LIN {X 0,Y 105.507,Z 842.039,A -85,B 0,C 180,E1 -26362.344,E2 -26362.344} C_VEL
LIN {X 0,Y 105.583,Z 840.616,A -85,B 0,C 180,E1 -26366.845,E2 -26366.845} C_VEL
LIN {X 0,Y 105.811,Z 839.235,A -85,B 0,C 180,E1 -26370,E2 -26370} C_VEL
LIN {X 0,Y 105.61,Z 835.784,A -85,B 0,C 180,E1 -26375.729,E2 -26375.729} C_VEL
LIN {X 0,Y 106.123,Z 831.156,A -85,B 0,C 180,E1 -26381.459,E2 -26381.459} C_VEL
LIN {X 0,Y 107.753,Z 824.08,A -85,B 0,C 180,E1 -26388.047,E2 -26388.047} C_VEL
LIN {X 0,Y 110.175,Z 816.366,A -85,B 0,C 180,E1 -26393.495,E2 -26393.495} C_VEL
LIN {X 0,Y 112.77,Z 808.397,A -85,B 0,C 180,E1 -26397.866,E2 -26397.866} C_VEL
LIN {X 0,Y 116.022,Z 799.047,A -85,B 0,C 180,E1 -26401.859,E2 -26401.859} C_VEL
LIN {X 0,Y 119.623,Z 788.064,A -85,B 0,C 180,E1 -26405.461,E2 -26405.461} C_VEL
LIN {X 0,Y 123.122,Z 776.115,A -85,B 0,C 180,E1 -26408.371,E2 -26408.371} C_VEL
LIN {X 0,Y 124.907,Z 768.802,A -85,B 0,C 180,E1 -26409.785,E2 -26409.785} C_VEL
LIN {X 0,Y 125.577,Z 763.379,A -85,B 0,C 180,E1 -26410.817,E2 -26410.817} C_VEL
LIN {X 0,Y 124.86,Z 754.314,A -85,B 0,C 180,E1 -26412.635,E2 -26412.635} C_VEL
LIN {X 0,Y 123.8,Z 745.016,A -85,B 0,C 180,E1 -26414.201,E2 -26414.201} C_VEL
LIN {X 0,Y 123.899,Z 739.222,A -85,B 0,C 180,E1 -26414.796,E2 -26414.796} C_VEL
LIN {X 0,Y 126.912,Z 703.597,A -85,B 0,C 180,E1 -26416.978,E2 -26416.978} C_VEL
LIN {X 0,Y 126.157,Z 693.57,A -85,B 0,C 180,E1 -26418.047,E2 -26418.047} C_VEL
LIN {X 0,Y 121.74,Z 679.502,A -85,B 0,C 180,E1 -26420.71,E2 -26420.71} C_VEL
LIN {X 0,Y 116.424,Z 665.324,A -85,B 0,C 180,E1 -26423.976,E2 -26423.976} C_VEL
LIN {X 0,Y 112.883,Z 657.742,A -85,B 0,C 180,E1 -26426.201,E2 -26426.201} C_VEL
LIN {X 0,Y 107.627,Z 649.272,A -85,B 0,C 180,E1 -26429.595,E2 -26429.595} C_VEL
LIN {X 0,Y 105.851,Z 646.479,A -85,B 0,C 180,E1 -26430.815,E2 -26430.815} C_VEL
LIN {X 0,Y 103.858,Z 643.285,A -85,B 0,C 180,E1 -26432.273,E2 -26432.273} C_VEL
LIN {X 0,Y 101.38,Z 640.128,A -85,B 0,C 180,E1 -26434.117,E2 -26434.117} C_VEL
LIN {X 0,Y 100.745,Z 637.925,A -85,B 0,C 180,E1 -26434.819,E2 -26434.819} C_VEL
LIN {X 0,Y 100.81,Z 637.922,A -85,B 0,C 180,E1 -26439.598,E2 -26439.598} C_VEL
LIN {X 0,Y 101.186,Z 637.873,A -85,B 0,C 180,E1 -26447.971,E2 -26447.971} C_VEL
LIN {X 0,Y 101.263,Z 637.855,A -85,B 0,C 180,E1 -26452.019,E2 -26452.019} C_VEL
LIN {X 0,Y 101.846,Z 637.775,A -85,B 0,C 180,E1 -26459.998,E2 -26459.998} C_VEL
LIN {X 0,Y 101.264,Z 637.869,A -85,B 0,C 180,E1 -26467.977,E2 -26467.977} C_VEL
LIN {X 0,Y 101.122,Z 637.858,A -85,B 0,C 180,E1 -26473.349,E2 -26473.349} C_VEL
LIN {X 0,Y 100.813,Z 637.923,A -85,B 0,C 180,E1 -26480.398,E2 -26480.398} C_VEL
LIN {X 0,Y 100.771,Z 637.901,A -85,B 0,C 180,E1 -26484.957,E2 -26484.957} C_VEL
LIN {X 0,Y 100.702,Z 637.938,A -85,B 0,C 180,E1 -26493.127,E2 -26493.127} C_VEL
LIN {X 0,Y 100.697,Z 637.919,A -85,B 0,C 180,E1 -26499.852,E2 -26499.852} C_VEL
LIN {X 0,Y 100.727,Z 637.934,A -85,B 0,C 180,E1 -26505.756,E2 -26505.756} C_VEL
LIN {X 0,Y 100.667,Z 637.925,A -85,B 0,C 180,E1 -26511.074,E2 -26511.074} C_VEL
LIN {X 0,Y 100.696,Z 637.935,A -85,B 0,C 180,E1 -26516.877,E2 -26516.877} C_VEL
LIN {X 0,Y 100.783,Z 637.928,A -85,B 0,C 180,E1 -26525.267,E2 -26525.267} C_VEL
LIN {X 0,Y 100.886,Z 638.058,A -85,B 0,C 180,E1 -26531.284,E2 -26531.284} C_VEL
LIN {X 0,Y 101.875,Z 640.799,A -85,B 0,C 180,E1 -26532.253,E2 -26532.253} C_VEL
LIN {X 0,Y 104.241,Z 643.451,A -85,B 0,C 180,E1 -26533.956,E2 -26533.956} C_VEL
LIN {X 0,Y 106.42,Z 646.692,A -85,B 0,C 180,E1 -26535.509,E2 -26535.509} C_VEL
LIN {X 0,Y 109.893,Z 651.957,A -85,B 0,C 180,E1 -26537.795,E2 -26537.795} C_VEL
LIN {X 0,Y 117.451,Z 664.633,A -85,B 0,C 180,E1 -26542.344,E2 -26542.344} C_VEL
LIN {X 0,Y 125.255,Z 682.339,A -85,B 0,C 180,E1 -26546.683,E2 -26546.683} C_VEL
LIN {X 0,Y 127.714,Z 688.733,A -85,B 0,C 180,E1 -26547.991,E2 -26547.991} C_VEL
LIN {X 0,Y 123.869,Z 730.785,A -85,B 0,C 180,E1 -26550.508,E2 -26550.508} C_VEL
LIN {X 0,Y 121.841,Z 745.154,A -85,B 0,C 180,E1 -26552.014,E2 -26552.014} C_VEL
LIN {X 0,Y 119.489,Z 756.549,A -85,B 0,C 180,E1 -26553.713,E2 -26553.713} C_VEL
LIN {X 0,Y 116.492,Z 768.644,A -85,B 0,C 180,E1 -26556.212,E2 -26556.212} C_VEL
LIN {X 0,Y 112.705,Z 781.046,A -85,B 0,C 180,E1 -26559.623,E2 -26559.623} C_VEL
LIN {X 0,Y 109.184,Z 791.561,A -85,B 0,C 180,E1 -26563.524,E2 -26563.524} C_VEL
LIN {X 0,Y 105.565,Z 801.658,A -85,B 0,C 180,E1 -26568.435,E2 -26568.435} C_VEL
LIN {X 0,Y 102.872,Z 809.142,A -85,B 0,C 180,E1 -26573.144,E2 -26573.144} C_VEL
LIN {X 0,Y 100.663,Z 815.792,A -85,B 0,C 180,E1 -26578.431,E2 -26578.431} C_VEL
LIN {X 0,Y 98.92,Z 821.873,A -85,B 0,C 180,E1 -26584.636,E2 -26584.636} C_VEL
LIN {X 0,Y 97.816,Z 827.335,A -85,B 0,C 180,E1 -26592.091,E2 -26592.091} C_VEL
LIN {X 0,Y 98.036,Z 831.381,A -85,B 0,C 180,E1 -26599.823,E2 -26599.823} C_VEL
LIN {X 0,Y 99.854,Z 833.955,A -85,B 0,C 180,E1 -26607.626,E2 -26607.626} C_VEL
LIN {X 0,Y 102.246,Z 834.975,A -85,B 0,C 180,E1 -26613.323,E2 -26613.323} C_VEL
LIN {X 0,Y 107.098,Z 835.004,A -85,B 0,C 180,E1 -26620.848,E2 -26620.848} C_VEL
LIN {X 0,Y 111.102,Z 834.19,A -85,B 0,C 180,E1 -26625.345,E2 -26625.345} C_VEL
LIN {X 0,Y 115.718,Z 832.693,A -85,B 0,C 180,E1 -26629.504,E2 -26629.504} C_VEL
LIN {X 0,Y 123.721,Z 829.106,A -85,B 0,C 180,E1 -26635.114,E2 -26635.114} C_VEL
LIN {X 0,Y 131.219,Z 824.778,A -85,B 0,C 180,E1 -26639.243,E2 -26639.243} C_VEL
LIN {X 0,Y 139.405,Z 819.061,A -85,B 0,C 180,E1 -26642.891,E2 -26642.891} C_VEL
LIN {X 0,Y 146.38,Z 813.354,A -85,B 0,C 180,E1 -26645.512,E2 -26645.512} C_VEL
LIN {X 0,Y 153.61,Z 806.471,A -85,B 0,C 180,E1 -26647.89,E2 -26647.89} C_VEL
LIN {X 0,Y 161.109,Z 798.113,A -85,B 0,C 180,E1 -26650.05,E2 -26650.05} C_VEL
LIN {X 0,Y 167.935,Z 789.141,A -85,B 0,C 180,E1 -26651.742,E2 -26651.742} C_VEL
LIN {X 0,Y 174.832,Z 778.191,A -85,B 0,C 180,E1 -26653.355,E2 -26653.355} C_VEL
LIN {X 0,Y 180.883,Z 766.378,A -85,B 0,C 180,E1 -26654.649,E2 -26654.649} C_VEL
LIN {X 0,Y 185.753,Z 754.041,A -85,B 0,C 180,E1 -26655.675,E2 -26655.675} C_VEL
LIN {X 0,Y 189.546,Z 741.072,A -85,B 0,C 180,E1 -26656.406,E2 -26656.406} C_VEL
LIN {X 0,Y 191.061,Z 734.083,A -85,B 0,C 180,E1 -26656.709,E2 -26656.709} C_VEL
LIN {X 0,Y 190.49,Z 732.621,A -85,B 0,C 180,E1 -26659.394,E2 -26659.394} C_VEL
LIN {X 0,Y 190.206,Z 732.592,A -85,B 0,C 180,E1 -26662.525,E2 -26662.525} C_VEL
LIN {X 0,Y 190.233,Z 735.09,A -85,B 0,C 180,E1 -26665.607,E2 -26665.607} C_VEL
LIN {X 0,Y 190.431,Z 736.832,A -85,B 0,C 180,E1 -26667.146,E2 -26667.146} C_VEL
LIN {X 0,Y 190.517,Z 737.806,A -85,B 0,C 180,E1 -26667.826,E2 -26667.826} C_VEL
LIN {X 0,Y 187.086,Z 751.386,A -85,B 0,C 180,E1 -26668.382,E2 -26668.382} C_VEL
LIN {X 0,Y 182.826,Z 763.398,A -85,B 0,C 180,E1 -26669.013,E2 -26669.013} C_VEL
LIN {X 0,Y 177.372,Z 775.257,A -85,B 0,C 180,E1 -26669.919,E2 -26669.919} C_VEL
LIN {X 0,Y 170.424,Z 787.344,A -85,B 0,C 180,E1 -26671.166,E2 -26671.166} C_VEL
LIN {X 0,Y 162.951,Z 798.092,A -85,B 0,C 180,E1 -26672.754,E2 -26672.754} C_VEL
LIN {X 0,Y 154.273,Z 808.469,A -85,B 0,C 180,E1 -26674.917,E2 -26674.917} C_VEL
LIN {X 0,Y 147.223,Z 815.602,A -85,B 0,C 180,E1 -26676.91,E2 -26676.91} C_VEL
LIN {X 0,Y 137.903,Z 823.753,A -85,B 0,C 180,E1 -26680.144,E2 -26680.144} C_VEL
LIN {X 0,Y 130.48,Z 829.369,A -85,B 0,C 180,E1 -26683.354,E2 -26683.354} C_VEL
LIN {X 0,Y 123.528,Z 833.895,A -85,B 0,C 180,E1 -26686.944,E2 -26686.944} C_VEL
LIN {X 0,Y 115.371,Z 838.364,A -85,B 0,C 180,E1 -26692.472,E2 -26692.472} C_VEL
LIN {X 0,Y 108.476,Z 841.336,A -85,B 0,C 180,E1 -26698.782,E2 -26698.782} C_VEL
LIN {X 0,Y 103.18,Z 842.778,A -85,B 0,C 180,E1 -26705.878,E2 -26705.878} C_VEL
LIN {X 0,Y 99.85,Z 842.798,A -85,B 0,C 180,E1 -26713.648,E2 -26713.648} C_VEL
LIN {X 0,Y 98.483,Z 841.375,A -85,B 0,C 180,E1 -26721.795,E2 -26721.795} C_VEL
LIN {X 0,Y 98.543,Z 839.693,A -85,B 0,C 180,E1 -26726.862,E2 -26726.862} C_VEL
LIN {X 0,Y 98.752,Z 838.329,A -85,B 0,C 180,E1 -26730,E2 -26730} C_VEL
LIN {X 0,Y 98.559,Z 834.707,A -85,B 0,C 180,E1 -26736.14,E2 -26736.14} C_VEL
LIN {X 0,Y 99.163,Z 829.901,A -85,B 0,C 180,E1 -26742.276,E2 -26742.276} C_VEL
LIN {X 0,Y 100.66,Z 823.745,A -85,B 0,C 180,E1 -26748.311,E2 -26748.311} C_VEL
LIN {X 0,Y 103.166,Z 816.036,A -85,B 0,C 180,E1 -26754.125,E2 -26754.125} C_VEL
LIN {X 0,Y 106.558,Z 806.291,A -85,B 0,C 180,E1 -26759.646,E2 -26759.646} C_VEL
LIN {X 0,Y 110.231,Z 796.046,A -85,B 0,C 180,E1 -26764.017,E2 -26764.017} C_VEL
LIN {X 0,Y 113.917,Z 785.002,A -85,B 0,C 180,E1 -26767.533,E2 -26767.533} C_VEL
LIN {X 0,Y 117.16,Z 774.095,A -85,B 0,C 180,E1 -26770.153,E2 -26770.153} C_VEL
LIN {X 0,Y 120.102,Z 762.182,A -85,B 0,C 180,E1 -26772.294,E2 -26772.294} C_VEL
LIN {X 0,Y 122.613,Z 748.643,A -85,B 0,C 180,E1 -26773.989,E2 -26773.989} C_VEL
LIN {X 0,Y 123.899,Z 739.222,A -85,B 0,C 180,E1 -26774.796,E2 -26774.796} C_VEL
LIN {X 0,Y 123.887,Z 733.426,A -85,B 0,C 180,E1 -26775.338,E2 -26775.338} C_VEL
LIN {X 0,Y 120.636,Z 714.621,A -85,B 0,C 180,E1 -26777.918,E2 -26777.918} C_VEL
LIN {X 0,Y 120.649,Z 708.81,A -85,B 0,C 180,E1 -26778.427,E2 -26778.427} C_VEL
LIN {X 0,Y 120.935,Z 703.551,A -85,B 0,C 180,E1 -26778.807,E2 -26778.807} C_VEL
LIN {X 0,Y 120.332,Z 695.575,A -85,B 0,C 180,E1 -26779.728,E2 -26779.728} C_VEL
LIN {X 0,Y 116.176,Z 682.158,A -85,B 0,C 180,E1 -26782.432,E2 -26782.432} C_VEL
LIN {X 0,Y 110.783,Z 667.555,A -85,B 0,C 180,E1 -26786.084,E2 -26786.084} C_VEL
LIN {X 0,Y 108.118,Z 661.9,A -85,B 0,C 180,E1 -26787.932,E2 -26787.932} C_VEL
LIN {X 0,Y 101.977,Z 651.808,A -85,B 0,C 180,E1 -26792.275,E2 -26792.275} C_VEL
LIN {X 0,Y 99.367,Z 647.874,A -85,B 0,C 180,E1 -26794.342,E2 -26794.342} C_VEL
LIN {X 0,Y 97.298,Z 644.843,A -85,B 0,C 180,E1 -26796.087,E2 -26796.087} C_VEL
LIN {X 0,Y 96.693,Z 643.761,A -85,B 0,C 180,E1 -26796.649,E2 -26796.649} C_VEL
LIN {X 0,Y 94.607,Z 641.473,A -85,B 0,C 180,E1 -26798.48,E2 -26798.48} C_VEL
LIN {X 0,Y 93.783,Z 638.795,A -85,B 0,C 180,E1 -26799.719,E2 -26799.719} C_VEL
LIN {X 0,Y 94.09,Z 638.764,A -85,B 0,C 180,E1 -26807.049,E2 -26807.049} C_VEL
LIN {X 0,Y 94.196,Z 638.732,A -85,B 0,C 180,E1 -26811.416,E2 -26811.416} C_VEL
LIN {X 0,Y 94.776,Z 638.654,A -85,B 0,C 180,E1 -26819.998,E2 -26819.998} C_VEL
LIN {X 0,Y 94.197,Z 638.747,A -85,B 0,C 180,E1 -26828.579,E2 -26828.579} C_VEL
LIN {X 0,Y 94.039,Z 638.739,A -85,B 0,C 180,E1 -26833.706,E2 -26833.706} C_VEL
LIN {X 0,Y 93.69,Z 638.801,A -85,B 0,C 180,E1 -26842.026,E2 -26842.026} C_VEL
LIN {X 0,Y 93.618,Z 638.792,A -85,B 0,C 180,E1 -26846.768,E2 -26846.768} C_VEL
LIN {X 0,Y 93.609,Z 638.815,A -85,B 0,C 180,E1 -26854.326,E2 -26854.326} C_VEL
LIN {X 0,Y 93.628,Z 638.819,A -85,B 0,C 180,E1 -26862.495,E2 -26862.495} C_VEL
LIN {X 0,Y 93.598,Z 638.802,A -85,B 0,C 180,E1 -26868.662,E2 -26868.662} C_VEL
LIN {X 0,Y 93.599,Z 638.825,A -85,B 0,C 180,E1 -26875.681,E2 -26875.681} C_VEL
LIN {X 0,Y 93.665,Z 638.818,A -85,B 0,C 180,E1 -26884.205,E2 -26884.205} C_VEL
LIN {X 0,Y 93.719,Z 638.857,A -85,B 0,C 180,E1 -26886.466,E2 -26886.466} C_VEL
LIN {X 0,Y 94.603,Z 641.463,A -85,B 0,C 180,E1 -26887.526,E2 -26887.526} C_VEL
LIN {X 0,Y 96.702,Z 643.724,A -85,B 0,C 180,E1 -26889.328,E2 -26889.328} C_VEL
LIN {X 0,Y 97.427,Z 644.758,A -85,B 0,C 180,E1 -26889.954,E2 -26889.954} C_VEL
LIN {X 0,Y 99.513,Z 647.872,A -85,B 0,C 180,E1 -26891.727,E2 -26891.727} C_VEL
LIN {X 0,Y 100.58,Z 649.179,A -85,B 0,C 180,E1 -26892.558,E2 -26892.558} C_VEL
LIN {X 0,Y 105.142,Z 655.973,A -85,B 0,C 180,E1 -26895.939,E2 -26895.939} C_VEL
LIN {X 0,Y 112.658,Z 668.93,A -85,B 0,C 180,E1 -26900.848,E2 -26900.848} C_VEL
LIN {X 0,Y 119.963,Z 685.957,A -85,B 0,C 180,E1 -26905.255,E2 -26905.255} C_VEL
LIN {X 0,Y 121.748,Z 691.098,A -85,B 0,C 180,E1 -26906.309,E2 -26906.309} C_VEL
LIN {X 0,Y 117.785,Z 731.396,A -85,B 0,C 180,E1 -26908.785,E2 -26908.785} C_VEL
LIN {X 0,Y 115.797,Z 744.729,A -85,B 0,C 180,E1 -26910.217,E2 -26910.217} C_VEL
LIN {X 0,Y 113.226,Z 756.797,A -85,B 0,C 180,E1 -26912.065,E2 -26912.065} C_VEL
LIN {X 0,Y 110.198,Z 768.519,A -85,B 0,C 180,E1 -26914.572,E2 -26914.572} C_VEL
LIN {X 0,Y 106.425,Z 780.27,A -85,B 0,C 180,E1 -26917.897,E2 -26917.897} C_VEL
LIN {X 0,Y 102.829,Z 790.679,A -85,B 0,C 180,E1 -26921.832,E2 -26921.832} C_VEL
LIN {X 0,Y 98.939,Z 801.026,A -85,B 0,C 180,E1 -26927.038,E2 -26927.038} C_VEL
LIN {X 0,Y 95.746,Z 809.537,A -85,B 0,C 180,E1 -26932.666,E2 -26932.666} C_VEL
LIN {X 0,Y 93.15,Z 817.199,A -85,B 0,C 180,E1 -26939.367,E2 -26939.367} C_VEL
LIN {X 0,Y 91.604,Z 822.513,A -85,B 0,C 180,E1 -26945.364,E2 -26945.364} C_VEL
LIN {X 0,Y 90.762,Z 826.881,A -85,B 0,C 180,E1 -26951.639,E2 -26951.639} C_VEL
LIN {X 0,Y 90.777,Z 830.425,A -85,B 0,C 180,E1 -26958.313,E2 -26958.313} C_VEL
LIN {X 0,Y 92.378,Z 833.555,A -85,B 0,C 180,E1 -26966.809,E2 -26966.809} C_VEL
LIN {X 0,Y 95.035,Z 835.066,A -85,B 0,C 180,E1 -26973.662,E2 -26973.662} C_VEL
LIN {X 0,Y 98.125,Z 835.577,A -85,B 0,C 180,E1 -26979.018,E2 -26979.018} C_VEL
LIN {X 0,Y 102.213,Z 835.342,A -85,B 0,C 180,E1 -26984.28,E2 -26984.28} C_VEL
LIN {X 0,Y 107.28,Z 834.296,A -85,B 0,C 180,E1 -26989.306,E2 -26989.306} C_VEL
LIN {X 0,Y 113.091,Z 832.418,A -85,B 0,C 180,E1 -26993.874,E2 -26993.874} C_VEL
LIN {X 0,Y 119.551,Z 829.672,A -85,B 0,C 180,E1 -26997.925,E2 -26997.925} C_VEL
LIN {X 0,Y 128.331,Z 824.95,A -85,B 0,C 180,E1 -27002.331,E2 -27002.331} C_VEL
LIN {X 0,Y 137.033,Z 819.188,A -85,B 0,C 180,E1 -27005.889,E2 -27005.889} C_VEL
LIN {X 0,Y 145.96,Z 812.026,A -85,B 0,C 180,E1 -27008.888,E2 -27008.888} C_VEL
LIN {X 0,Y 155.535,Z 802.716,A -85,B 0,C 180,E1 -27011.619,E2 -27011.619} C_VEL
LIN {X 0,Y 162.888,Z 794.206,A -85,B 0,C 180,E1 -27013.39,E2 -27013.39} C_VEL
LIN {X 0,Y 170.093,Z 784.173,A -85,B 0,C 180,E1 -27014.968,E2 -27014.968} C_VEL
LIN {X 0,Y 176.246,Z 773.773,A -85,B 0,C 180,E1 -27016.21,E2 -27016.21} C_VEL
LIN {X 0,Y 181.857,Z 762.003,A -85,B 0,C 180,E1 -27017.284,E2 -27017.284} C_VEL
LIN {X 0,Y 186.117,Z 750.546,A -85,B 0,C 180,E1 -27018.084,E2 -27018.084} C_VEL
LIN {X 0,Y 189.08,Z 739.923,A -85,B 0,C 180,E1 -27018.664,E2 -27018.664} C_VEL
LIN {X 0,Y 188.982,Z 739.555,A -85,B 0,C 180,E1 -27019.555,E2 -27019.555} C_VEL
LIN {X 0,Y 188.748,Z 739.568,A -85,B 0,C 180,E1 -27022.51,E2 -27022.51} C_VEL
LIN {X 0,Y 188.622,Z 742.467,A -85,B 0,C 180,E1 -27025.859,E2 -27025.859} C_VEL
LIN {X 0,Y 184.48,Z 756.22,A -85,B 0,C 180,E1 -27026.42,E2 -27026.42} C_VEL
LIN {X 0,Y 179.622,Z 768.209,A -85,B 0,C 180,E1 -27027.113,E2 -27027.113} C_VEL
LIN {X 0,Y 173.247,Z 780.405,A -85,B 0,C 180,E1 -27028.079,E2 -27028.079} C_VEL
LIN {X 0,Y 166.211,Z 791.358,A -85,B 0,C 180,E1 -27029.299,E2 -27029.299} C_VEL
LIN {X 0,Y 159.316,Z 800.338,A -85,B 0,C 180,E1 -27030.662,E2 -27030.662} C_VEL
LIN {X 0,Y 150.398,Z 810.137,A -85,B 0,C 180,E1 -27032.743,E2 -27032.743} C_VEL
LIN {X 0,Y 141.745,Z 818.173,A -85,B 0,C 180,E1 -27035.107,E2 -27035.107} C_VEL
LIN {X 0,Y 133.482,Z 824.729,A -85,B 0,C 180,E1 -27037.838,E2 -27037.838} C_VEL
LIN {X 0,Y 125.751,Z 830.037,A -85,B 0,C 180,E1 -27041.021,E2 -27041.021} C_VEL
LIN {X 0,Y 118.45,Z 834.317,A -85,B 0,C 180,E1 -27044.604,E2 -27044.604} C_VEL
LIN {X 0,Y 109.815,Z 838.571,A -85,B 0,C 180,E1 -27050.21,E2 -27050.21} C_VEL
LIN {X 0,Y 102.46,Z 841.237,A -85,B 0,C 180,E1 -27056.72,E2 -27056.72} C_VEL
LIN {X 0,Y 96.739,Z 842.474,A -85,B 0,C 180,E1 -27064.159,E2 -27064.159} C_VEL
LIN {X 0,Y 93.023,Z 842.298,A -85,B 0,C 180,E1 -27072.41,E2 -27072.41} C_VEL
LIN {X 0,Y 91.467,Z 840.637,A -85,B 0,C 180,E1 -27081.16,E2 -27081.16} C_VEL
LIN {X 0,Y 91.509,Z 838.797,A -85,B 0,C 180,E1 -27086.809,E2 -27086.809} C_VEL
LIN {X 0,Y 91.695,Z 837.408,A -85,B 0,C 180,E1 -27090,E2 -27090} C_VEL
LIN {X 0,Y 91.519,Z 833.589,A -85,B 0,C 180,E1 -27096.614,E2 -27096.614} C_VEL
LIN {X 0,Y 92.239,Z 828.574,A -85,B 0,C 180,E1 -27103.213,E2 -27103.213} C_VEL
LIN {X 0,Y 93.948,Z 822.181,A -85,B 0,C 180,E1 -27109.671,E2 -27109.671} C_VEL
LIN {X 0,Y 96.695,Z 814.135,A -85,B 0,C 180,E1 -27115.854,E2 -27115.854} C_VEL
LIN {X 0,Y 99.745,Z 805.915,A -85,B 0,C 180,E1 -27120.719,E2 -27120.719} C_VEL
LIN {X 0,Y 103.507,Z 795.936,A -85,B 0,C 180,E1 -27125.242,E2 -27125.242} C_VEL
LIN {X 0,Y 107.442,Z 784.692,A -85,B 0,C 180,E1 -27129.019,E2 -27129.019} C_VEL
LIN {X 0,Y 110.827,Z 773.799,A -85,B 0,C 180,E1 -27131.746,E2 -27131.746} C_VEL
LIN {X 0,Y 114.175,Z 760.719,A -85,B 0,C 180,E1 -27134.133,E2 -27134.133} C_VEL
LIN {X 0,Y 116.664,Z 747.345,A -85,B 0,C 180,E1 -27135.826,E2 -27135.826} C_VEL
LIN {X 0,Y 118.395,Z 733.513,A -85,B 0,C 180,E1 -27136.919,E2 -27136.919} C_VEL
LIN {X 0,Y 120.649,Z 708.81,A -85,B 0,C 180,E1 -27138.427,E2 -27138.427} C_VEL
LIN {X 0,Y 120.572,Z 705.009,A -85,B 0,C 180,E1 -27138.795,E2 -27138.795} C_VEL
LIN {X 0,Y 119.745,Z 701.405,A -85,B 0,C 180,E1 -27139.393,E2 -27139.393} C_VEL
LIN {X 0,Y 118.4,Z 698.014,A -85,B 0,C 180,E1 -27140.164,E2 -27140.164} C_VEL
LIN {X 0,Y 110.38,Z 683.673,A -85,B 0,C 180,E1 -27144.553,E2 -27144.553} C_VEL
LIN {X 0,Y 109.72,Z 681.909,A -85,B 0,C 180,E1 -27145.018,E2 -27145.018} C_VEL
LIN {X 0,Y 104.964,Z 669.063,A -85,B 0,C 180,E1 -27148.633,E2 -27148.633} C_VEL
LIN {X 0,Y 99.77,Z 659.846,A -85,B 0,C 180,E1 -27152.528,E2 -27152.528} C_VEL
LIN {X 0,Y 95.437,Z 652.984,A -85,B 0,C 180,E1 -27156.218,E2 -27156.218} C_VEL
LIN {X 0,Y 92.964,Z 649.251,A -85,B 0,C 180,E1 -27158.517,E2 -27158.517} C_VEL
LIN {X 0,Y 90.71,Z 646.109,A -85,B 0,C 180,E1 -27160.773,E2 -27160.773} C_VEL
LIN {X 0,Y 90.069,Z 644.86,A -85,B 0,C 180,E1 -27161.516,E2 -27161.516} C_VEL
LIN {X 0,Y 87.854,Z 642.603,A -85,B 0,C 180,E1 -27163.905,E2 -27163.905} C_VEL
LIN {X 0,Y 86.916,Z 639.892,A -85,B 0,C 180,E1 -27165.312,E2 -27165.312} C_VEL
LIN {X 0,Y 86.969,Z 639.655,A -85,B 0,C 180,E1 -27165.968,E2 -27165.968} C_VEL
LIN {X 0,Y 87.105,Z 639.614,A -85,B 0,C 180,E1 -27170.711,E2 -27170.711} C_VEL
LIN {X 0,Y 87.706,Z 639.534,A -85,B 0,C 180,E1 -27179.998,E2 -27179.998} C_VEL
LIN {X 0,Y 87.105,Z 639.625,A -85,B 0,C 180,E1 -27189.284,E2 -27189.284} C_VEL
LIN {X 0,Y 86.948,Z 639.623,A -85,B 0,C 180,E1 -27194.085,E2 -27194.085} C_VEL
LIN {X 0,Y 86.659,Z 639.687,A -85,B 0,C 180,E1 -27198.927,E2 -27198.927} C_VEL
LIN {X 0,Y 86.581,Z 639.668,A -85,B 0,C 180,E1 -27206.763,E2 -27206.763} C_VEL
LIN {X 0,Y 86.534,Z 639.683,A -85,B 0,C 180,E1 -27215.693,E2 -27215.693} C_VEL
LIN {X 0,Y 86.553,Z 639.702,A -85,B 0,C 180,E1 -27223.049,E2 -27223.049} C_VEL
LIN {X 0,Y 86.505,Z 639.683,A -85,B 0,C 180,E1 -27229.463,E2 -27229.463} C_VEL
LIN {X 0,Y 86.545,Z 639.705,A -85,B 0,C 180,E1 -27235.359,E2 -27235.359} C_VEL
LIN {X 0,Y 86.494,Z 639.814,A -85,B 0,C 180,E1 -27240.238,E2 -27240.238} C_VEL
LIN {X 0,Y 87.41,Z 642.419,A -85,B 0,C 180,E1 -27241.619,E2 -27241.619} C_VEL
LIN {X 0,Y 89.42,Z 644.526,A -85,B 0,C 180,E1 -27243.853,E2 -27243.853} C_VEL
LIN {X 0,Y 90.277,Z 645.19,A -85,B 0,C 180,E1 -27244.708,E2 -27244.708} C_VEL
LIN {X 0,Y 92.207,Z 648.436,A -85,B 0,C 180,E1 -27246.795,E2 -27246.795} C_VEL
LIN {X 0,Y 93.86,Z 650.398,A -85,B 0,C 180,E1 -27248.323,E2 -27248.323} C_VEL
LIN {X 0,Y 97.533,Z 655.716,A -85,B 0,C 180,E1 -27251.529,E2 -27251.529} C_VEL
LIN {X 0,Y 100.981,Z 660.89,A -85,B 0,C 180,E1 -27254.292,E2 -27254.292} C_VEL
LIN {X 0,Y 107.991,Z 673.429,A -85,B 0,C 180,E1 -27259.274,E2 -27259.274} C_VEL
LIN {X 0,Y 114.654,Z 689.462,A -85,B 0,C 180,E1 -27263.703,E2 -27263.703} C_VEL
LIN {X 0,Y 115.771,Z 692.545,A -85,B 0,C 180,E1 -27264.411,E2 -27264.411} C_VEL
LIN {X 0,Y 111.744,Z 732.209,A -85,B 0,C 180,E1 -27266.958,E2 -27266.958} C_VEL
LIN {X 0,Y 109.669,Z 745.169,A -85,B 0,C 180,E1 -27268.393,E2 -27268.393} C_VEL
LIN {X 0,Y 106.957,Z 757.273,A -85,B 0,C 180,E1 -27270.312,E2 -27270.312} C_VEL
LIN {X 0,Y 103.775,Z 768.917,A -85,B 0,C 180,E1 -27272.901,E2 -27272.901} C_VEL
LIN {X 0,Y 99.81,Z 780.816,A -85,B 0,C 180,E1 -27276.439,E2 -27276.439} C_VEL
LIN {X 0,Y 96.046,Z 791.091,A -85,B 0,C 180,E1 -27280.54,E2 -27280.54} C_VEL
LIN {X 0,Y 91.938,Z 801.492,A -85,B 0,C 180,E1 -27286.114,E2 -27286.114} C_VEL
LIN {X 0,Y 88.48,Z 810.434,A -85,B 0,C 180,E1 -27292.524,E2 -27292.524} C_VEL
LIN {X 0,Y 85.946,Z 817.595,A -85,B 0,C 180,E1 -27299.381,E2 -27299.381} C_VEL
LIN {X 0,Y 84.406,Z 822.712,A -85,B 0,C 180,E1 -27305.65,E2 -27305.65} C_VEL
LIN {X 0,Y 83.639,Z 826.97,A -85,B 0,C 180,E1 -27312.238,E2 -27312.238} C_VEL
LIN {X 0,Y 84.082,Z 831.492,A -85,B 0,C 180,E1 -27321.755,E2 -27321.755} C_VEL
LIN {X 0,Y 86.492,Z 834.395,A -85,B 0,C 180,E1 -27330.824,E2 -27330.824} C_VEL
LIN {X 0,Y 90.405,Z 835.764,A -85,B 0,C 180,E1 -27338.883,E2 -27338.883} C_VEL
LIN {X 0,Y 94.704,Z 835.958,A -85,B 0,C 180,E1 -27344.733,E2 -27344.733} C_VEL
LIN {X 0,Y 102.172,Z 834.842,A -85,B 0,C 180,E1 -27352.095,E2 -27352.095} C_VEL
LIN {X 0,Y 107.791,Z 833.297,A -85,B 0,C 180,E1 -27356.264,E2 -27356.264} C_VEL
LIN {X 0,Y 116.995,Z 829.686,A -85,B 0,C 180,E1 -27361.611,E2 -27361.611} C_VEL
LIN {X 0,Y 127.227,Z 824.381,A -85,B 0,C 180,E1 -27366.126,E2 -27366.126} C_VEL
LIN {X 0,Y 135.199,Z 819.222,A -85,B 0,C 180,E1 -27369.016,E2 -27369.016} C_VEL
LIN {X 0,Y 145.246,Z 811.395,A -85,B 0,C 180,E1 -27372.031,E2 -27372.031} C_VEL
LIN {X 0,Y 154.179,Z 802.972,A -85,B 0,C 180,E1 -27374.29,E2 -27374.29} C_VEL
LIN {X 0,Y 161.612,Z 794.605,A -85,B 0,C 180,E1 -27375.894,E2 -27375.894} C_VEL
LIN {X 0,Y 169.444,Z 783.961,A -85,B 0,C 180,E1 -27377.457,E2 -27377.457} C_VEL
LIN {X 0,Y 176.022,Z 773.076,A -85,B 0,C 180,E1 -27378.629,E2 -27378.629} C_VEL
LIN {X 0,Y 181.681,Z 761.35,A -85,B 0,C 180,E1 -27379.615,E2 -27379.615} C_VEL
LIN {X 0,Y 185.783,Z 750.33,A -85,B 0,C 180,E1 -27380.313,E2 -27380.313} C_VEL
LIN {X 0,Y 187.019,Z 746.321,A -85,B 0,C 180,E1 -27380.577,E2 -27380.577} C_VEL
LIN {X 0,Y 186.93,Z 746.359,A -85,B 0,C 180,E1 -27382.085,E2 -27382.085} C_VEL
LIN {X 0,Y 186.816,Z 746.986,A -85,B 0,C 180,E1 -27382.965,E2 -27382.965} C_VEL
LIN {X 0,Y 186.596,Z 748.107,A -85,B 0,C 180,E1 -27383.898,E2 -27383.898} C_VEL
LIN {X 0,Y 182.032,Z 760.983,A -85,B 0,C 180,E1 -27384.44,E2 -27384.44} C_VEL
LIN {X 0,Y 176.601,Z 772.704,A -85,B 0,C 180,E1 -27385.132,E2 -27385.132} C_VEL
LIN {X 0,Y 169.301,Z 785.058,A -85,B 0,C 180,E1 -27386.146,E2 -27386.146} C_VEL
LIN {X 0,Y 162.156,Z 795.047,A -85,B 0,C 180,E1 -27387.319,E2 -27387.319} C_VEL
LIN {X 0,Y 154.375,Z 804.217,A -85,B 0,C 180,E1 -27388.796,E2 -27388.796} C_VEL
LIN {X 0,Y 145.24,Z 813.218,A -85,B 0,C 180,E1 -27390.809,E2 -27390.809} C_VEL
LIN {X 0,Y 136.407,Z 820.55,A -85,B 0,C 180,E1 -27393.153,E2 -27393.153} C_VEL
LIN {X 0,Y 126.552,Z 827.482,A -85,B 0,C 180,E1 -27396.368,E2 -27396.368} C_VEL
LIN {X 0,Y 118.606,Z 832.183,A -85,B 0,C 180,E1 -27399.619,E2 -27399.619} C_VEL
LIN {X 0,Y 111.188,Z 835.883,A -85,B 0,C 180,E1 -27403.375,E2 -27403.375} C_VEL
LIN {X 0,Y 104.245,Z 838.768,A -85,B 0,C 180,E1 -27407.871,E2 -27407.871} C_VEL
LIN {X 0,Y 96.595,Z 841.138,A -85,B 0,C 180,E1 -27414.406,E2 -27414.406} C_VEL
LIN {X 0,Y 90.4,Z 842.159,A -85,B 0,C 180,E1 -27422.196,E2 -27422.196} C_VEL
LIN {X 0,Y 86.256,Z 841.716,A -85,B 0,C 180,E1 -27430.979,E2 -27430.979} C_VEL
LIN {X 0,Y 84.477,Z 839.863,A -85,B 0,C 180,E1 -27440.422,E2 -27440.422} C_VEL
LIN {X 0,Y 84.476,Z 837.799,A -85,B 0,C 180,E1 -27446.742,E2 -27446.742} C_VEL
LIN {X 0,Y 84.64,Z 836.432,A -85,B 0,C 180,E1 -27450,E2 -27450} C_VEL
LIN {X 0,Y 84.509,Z 832.427,A -85,B 0,C 180,E1 -27457.166,E2 -27457.166} C_VEL
LIN {X 0,Y 85.594,Z 826.158,A -85,B 0,C 180,E1 -27465.477,E2 -27465.477} C_VEL
LIN {X 0,Y 87.746,Z 819.266,A -85,B 0,C 180,E1 -27472.361,E2 -27472.361} C_VEL
LIN {X 0,Y 90.337,Z 812.178,A -85,B 0,C 180,E1 -27477.825,E2 -27477.825} C_VEL
LIN {X 0,Y 93.725,Z 803.621,A -85,B 0,C 180,E1 -27482.931,E2 -27482.931} C_VEL
LIN {X 0,Y 97.808,Z 793.107,A -85,B 0,C 180,E1 -27487.637,E2 -27487.637} C_VEL
LIN {X 0,Y 101.53,Z 782.738,A -85,B 0,C 180,E1 -27491.116,E2 -27491.116} C_VEL
LIN {X 0,Y 105.136,Z 771.513,A -85,B 0,C 180,E1 -27493.909,E2 -27493.909} C_VEL
LIN {X 0,Y 108.357,Z 758.907,A -85,B 0,C 180,E1 -27496.182,E2 -27496.182} C_VEL
LIN {X 0,Y 110.833,Z 745.918,A -85,B 0,C 180,E1 -27497.825,E2 -27497.825} C_VEL
LIN {X 0,Y 112.49,Z 732.469,A -85,B 0,C 180,E1 -27498.891,E2 -27498.891} C_VEL
LIN {X 0,Y 115.06,Z 704.596,A -85,B 0,C 180,E1 -27500.679,E2 -27500.679} C_VEL
LIN {X 0,Y 114.624,Z 697.867,A -85,B 0,C 180,E1 -27501.483,E2 -27501.483} C_VEL
LIN {X 0,Y 110.368,Z 683.84,A -85,B 0,C 180,E1 -27504.54,E2 -27504.54} C_VEL
LIN {X 0,Y 109.72,Z 681.909,A -85,B 0,C 180,E1 -27505.018,E2 -27505.018} C_VEL
LIN {X 0,Y 107.504,Z 677.233,A -85,B 0,C 180,E1 -27506.514,E2 -27506.514} C_VEL
LIN {X 0,Y 104.576,Z 673.318,A -85,B 0,C 180,E1 -27508.345,E2 -27508.345} C_VEL
LIN {X 0,Y 94.062,Z 661.932,A -85,B 0,C 180,E1 -27515.877,E2 -27515.877} C_VEL
LIN {X 0,Y 89.49,Z 654.791,A -85,B 0,C 180,E1 -27520.351,E2 -27520.351} C_VEL
LIN {X 0,Y 87.111,Z 651.088,A -85,B 0,C 180,E1 -27523.068,E2 -27523.068} C_VEL
LIN {X 0,Y 84.527,Z 647.786,A -85,B 0,C 180,E1 -27526.25,E2 -27526.25} C_VEL
LIN {X 0,Y 83.55,Z 645.868,A -85,B 0,C 180,E1 -27527.674,E2 -27527.674} C_VEL
LIN {X 0,Y 81.381,Z 643.831,A -85,B 0,C 180,E1 -27530.679,E2 -27530.679} C_VEL
LIN {X 0,Y 80.239,Z 641.5,A -85,B 0,C 180,E1 -27532.764,E2 -27532.764} C_VEL
LIN {X 0,Y 80.055,Z 640.503,A -85,B 0,C 180,E1 -27533.381,E2 -27533.381} C_VEL
LIN {X 0,Y 80.637,Z 640.414,A -85,B 0,C 180,E1 -27539.997,E2 -27539.997} C_VEL
LIN {X 0,Y 79.99,Z 640.501,A -85,B 0,C 180,E1 -27550.118,E2 -27550.118} C_VEL
LIN {X 0,Y 79.763,Z 640.522,A -85,B 0,C 180,E1 -27555.325,E2 -27555.325} C_VEL
LIN {X 0,Y 79.519,Z 640.573,A -85,B 0,C 180,E1 -27560.7,E2 -27560.7} C_VEL
LIN {X 0,Y 79.48,Z 640.557,A -85,B 0,C 180,E1 -27567.843,E2 -27567.843} C_VEL
LIN {X 0,Y 79.444,Z 640.558,A -85,B 0,C 180,E1 -27577.235,E2 -27577.235} C_VEL
LIN {X 0,Y 79.463,Z 640.585,A -85,B 0,C 180,E1 -27585.032,E2 -27585.032} C_VEL
LIN {X 0,Y 79.42,Z 640.719,A -85,B 0,C 180,E1 -27591.813,E2 -27591.813} C_VEL
LIN {X 0,Y 80.226,Z 643.043,A -85,B 0,C 180,E1 -27593.577,E2 -27593.577} C_VEL
LIN {X 0,Y 82.617,Z 645.624,A -85,B 0,C 180,E1 -27597.23,E2 -27597.23} C_VEL
LIN {X 0,Y 83.471,Z 646.222,A -85,B 0,C 180,E1 -27598.33,E2 -27598.33} C_VEL
LIN {X 0,Y 85.083,Z 649.145,A -85,B 0,C 180,E1 -27600.604,E2 -27600.604} C_VEL
LIN {X 0,Y 87.31,Z 651.486,A -85,B 0,C 180,E1 -27603.166,E2 -27603.166} C_VEL
LIN {X 0,Y 89.77,Z 655.097,A -85,B 0,C 180,E1 -27605.927,E2 -27605.927} C_VEL
LIN {X 0,Y 95.39,Z 663.348,A -85,B 0,C 180,E1 -27611.215,E2 -27611.215} C_VEL
LIN {X 0,Y 102.913,Z 676.765,A -85,B 0,C 180,E1 -27617.255,E2 -27617.255} C_VEL
LIN {X 0,Y 109.463,Z 692.987,A -85,B 0,C 180,E1 -27622.014,E2 -27622.014} C_VEL
LIN {X 0,Y 109.867,Z 694.16,A -85,B 0,C 180,E1 -27622.304,E2 -27622.304} C_VEL
LIN {X 0,Y 105.834,Z 732.868,A -85,B 0,C 180,E1 -27624.905,E2 -27624.905} C_VEL
LIN {X 0,Y 103.663,Z 745.613,A -85,B 0,C 180,E1 -27626.356,E2 -27626.356} C_VEL
LIN {X 0,Y 100.62,Z 758.485,A -85,B 0,C 180,E1 -27628.499,E2 -27628.499} C_VEL
LIN {X 0,Y 96.777,Z 771.356,A -85,B 0,C 180,E1 -27631.565,E2 -27631.565} C_VEL
LIN {X 0,Y 92.821,Z 782.533,A -85,B 0,C 180,E1 -27635.217,E2 -27635.217} C_VEL
LIN {X 0,Y 88.794,Z 792.677,A -85,B 0,C 180,E1 -27639.683,E2 -27639.683} C_VEL
LIN {X 0,Y 84.58,Z 802.806,A -85,B 0,C 180,E1 -27645.667,E2 -27645.667} C_VEL
LIN {X 0,Y 81.563,Z 810.236,A -85,B 0,C 180,E1 -27651.481,E2 -27651.481} C_VEL
LIN {X 0,Y 78.978,Z 817.221,A -85,B 0,C 180,E1 -27658.553,E2 -27658.553} C_VEL
LIN {X 0,Y 77.02,Z 823.72,A -85,B 0,C 180,E1 -27667.31,E2 -27667.31} C_VEL
LIN {X 0,Y 76.458,Z 827.978,A -85,B 0,C 180,E1 -27674.817,E2 -27674.817} C_VEL
LIN {X 0,Y 77.467,Z 832.162,A -85,B 0,C 180,E1 -27684.734,E2 -27684.734} C_VEL
LIN {X 0,Y 80.441,Z 834.861,A -85,B 0,C 180,E1 -27694.1,E2 -27694.1} C_VEL
LIN {X 0,Y 83.677,Z 835.938,A -85,B 0,C 180,E1 -27700.372,E2 -27700.372} C_VEL
LIN {X 0,Y 87.888,Z 836.361,A -85,B 0,C 180,E1 -27706.122,E2 -27706.122} C_VEL
LIN {X 0,Y 92.738,Z 836.122,A -85,B 0,C 180,E1 -27711.285,E2 -27711.285} C_VEL
LIN {X 0,Y 98.615,Z 835.129,A -85,B 0,C 180,E1 -27716.124,E2 -27716.124} C_VEL
LIN {X 0,Y 108.22,Z 832.398,A -85,B 0,C 180,E1 -27722.141,E2 -27722.141} C_VEL
LIN {X 0,Y 118.261,Z 828.206,A -85,B 0,C 180,E1 -27726.828,E2 -27726.828} C_VEL
LIN {X 0,Y 128.714,Z 822.59,A -85,B 0,C 180,E1 -27730.64,E2 -27730.64} C_VEL
LIN {X 0,Y 137.119,Z 817.009,A -85,B 0,C 180,E1 -27733.141,E2 -27733.141} C_VEL
LIN {X 0,Y 145.761,Z 810.165,A -85,B 0,C 180,E1 -27735.358,E2 -27735.358} C_VEL
LIN {X 0,Y 154.568,Z 801.843,A -85,B 0,C 180,E1 -27737.289,E2 -27737.289} C_VEL
LIN {X 0,Y 163.469,Z 791.686,A -85,B 0,C 180,E1 -27738.947,E2 -27738.947} C_VEL
LIN {X 0,Y 170.607,Z 781.773,A -85,B 0,C 180,E1 -27740.172,E2 -27740.172} C_VEL
LIN {X 0,Y 176.972,Z 770.886,A -85,B 0,C 180,E1 -27741.192,E2 -27741.192} C_VEL
LIN {X 0,Y 181.833,Z 760.595,A -85,B 0,C 180,E1 -27741.937,E2 -27741.937} C_VEL
LIN {X 0,Y 182.095,Z 759.994,A -85,B 0,C 180,E1 -27742.141,E2 -27742.141} C_VEL
LIN {X 0,Y 176.767,Z 771.468,A -85,B 0,C 180,E1 -27742.733,E2 -27742.733} C_VEL
LIN {X 0,Y 169.657,Z 783.547,A -85,B 0,C 180,E1 -27743.581,E2 -27743.581} C_VEL
LIN {X 0,Y 162.326,Z 793.69,A -85,B 0,C 180,E1 -27744.607,E2 -27744.607} C_VEL
LIN {X 0,Y 154.312,Z 802.96,A -85,B 0,C 180,E1 -27745.911,E2 -27745.911} C_VEL
LIN {X 0,Y 144.886,Z 812.122,A -85,B 0,C 180,E1 -27747.72,E2 -27747.72} C_VEL
LIN {X 0,Y 135.69,Z 819.594,A -85,B 0,C 180,E1 -27749.826,E2 -27749.826} C_VEL
LIN {X 0,Y 125.354,Z 826.594,A -85,B 0,C 180,E1 -27752.759,E2 -27752.759} C_VEL
LIN {X 0,Y 116.977,Z 831.35,A -85,B 0,C 180,E1 -27755.8,E2 -27755.8} C_VEL
LIN {X 0,Y 108.971,Z 835.161,A -85,B 0,C 180,E1 -27759.294,E2 -27759.294} C_VEL
LIN {X 0,Y 99.311,Z 838.823,A -85,B 0,C 180,E1 -27764.955,E2 -27764.955} C_VEL
LIN {X 0,Y 90.91,Z 841.013,A -85,B 0,C 180,E1 -27771.798,E2 -27771.798} C_VEL
LIN {X 0,Y 84.183,Z 841.759,A -85,B 0,C 180,E1 -27779.941,E2 -27779.941} C_VEL
LIN {X 0,Y 79.554,Z 841.121,A -85,B 0,C 180,E1 -27789.307,E2 -27789.307} C_VEL
LIN {X 0,Y 77.512,Z 839.063,A -85,B 0,C 180,E1 -27799.552,E2 -27799.552} C_VEL
LIN {X 0,Y 77.448,Z 836.774,A -85,B 0,C 180,E1 -27806.602,E2 -27806.602} C_VEL
LIN {X 0,Y 77.597,Z 835.362,A -85,B 0,C 180,E1 -27810,E2 -27810} C_VEL
LIN {X 0,Y 77.517,Z 831.154,A -85,B 0,C 180,E1 -27817.816,E2 -27817.816} C_VEL
LIN {X 0,Y 78.514,Z 825.689,A -85,B 0,C 180,E1 -27825.577,E2 -27825.577} C_VEL
LIN {X 0,Y 80.74,Z 818.802,A -85,B 0,C 180,E1 -27833.06,E2 -27833.06} C_VEL
LIN {X 0,Y 83.468,Z 811.718,A -85,B 0,C 180,E1 -27838.956,E2 -27838.956} C_VEL
LIN {X 0,Y 87.051,Z 803.136,A -85,B 0,C 180,E1 -27844.411,E2 -27844.411} C_VEL
LIN {X 0,Y 91.033,Z 793.39,A -85,B 0,C 180,E1 -27849.064,E2 -27849.064} C_VEL
LIN {X 0,Y 95.267,Z 782.191,A -85,B 0,C 180,E1 -27853.029,E2 -27853.029} C_VEL
LIN {X 0,Y 99.047,Z 770.898,A -85,B 0,C 180,E1 -27855.924,E2 -27855.924} C_VEL
LIN {X 0,Y 102.403,Z 758.202,A -85,B 0,C 180,E1 -27858.274,E2 -27858.274} C_VEL
LIN {X 0,Y 105,Z 745.081,A -85,B 0,C 180,E1 -27859.954,E2 -27859.954} C_VEL
LIN {X 0,Y 106.91,Z 729.875,A -85,B 0,C 180,E1 -27861.129,E2 -27861.129} C_VEL
LIN {X 0,Y 109.277,Z 705.445,A -85,B 0,C 180,E1 -27862.739,E2 -27862.739} C_VEL
LIN {X 0,Y 108.9,Z 699.726,A -85,B 0,C 180,E1 -27863.488,E2 -27863.488} C_VEL
LIN {X 0,Y 104.993,Z 686.378,A -85,B 0,C 180,E1 -27866.658,E2 -27866.658} C_VEL
LIN {X 0,Y 100.292,Z 673.232,A -85,B 0,C 180,E1 -27870.532,E2 -27870.532} C_VEL
LIN {X 0,Y 95.738,Z 664.824,A -85,B 0,C 180,E1 -27874.348,E2 -27874.348} C_VEL
LIN {X 0,Y 94.062,Z 661.932,A -85,B 0,C 180,E1 -27875.877,E2 -27875.877} C_VEL
LIN {X 0,Y 92.07,Z 659.911,A -85,B 0,C 180,E1 -27877.561,E2 -27877.561} C_VEL
LIN {X 0,Y 88.27,Z 658.103,A -85,B 0,C 180,E1 -27880.836,E2 -27880.836} C_VEL
LIN {X 0,Y 83.89,Z 656.302,A -85,B 0,C 180,E1 -27885.256,E2 -27885.256} C_VEL
LIN {X 0,Y 82.646,Z 655.267,A -85,B 0,C 180,E1 -27886.746,E2 -27886.746} C_VEL
LIN {X 0,Y 80.662,Z 651.935,A -85,B 0,C 180,E1 -27889.735,E2 -27889.735} C_VEL
LIN {X 0,Y 78.514,Z 649.342,A -85,B 0,C 180,E1 -27893.25,E2 -27893.25} C_VEL
LIN {X 0,Y 77.563,Z 647.093,A -85,B 0,C 180,E1 -27895.334,E2 -27895.334} C_VEL
LIN {X 0,Y 75.412,Z 645.319,A -85,B 0,C 180,E1 -27899.663,E2 -27899.663} C_VEL
LIN {X 0,Y 73.332,Z 642.653,A -85,B 0,C 180,E1 -27905.497,E2 -27905.497} C_VEL
LIN {X 0,Y 72.949,Z 641.396,A -85,B 0,C 180,E1 -27907.609,E2 -27907.609} C_VEL
LIN {X 0,Y 72.755,Z 641.392,A -85,B 0,C 180,E1 -27914.993,E2 -27914.993} C_VEL
LIN {X 0,Y 72.396,Z 641.441,A -85,B 0,C 180,E1 -27922.846,E2 -27922.846} C_VEL
LIN {X 0,Y 72.374,Z 641.45,A -85,B 0,C 180,E1 -27929.08,E2 -27929.08} C_VEL
LIN {X 0,Y 72.413,Z 641.552,A -85,B 0,C 180,E1 -27937.045,E2 -27937.045} C_VEL
LIN {X 0,Y 73.156,Z 644.092,A -85,B 0,C 180,E1 -27940.644,E2 -27940.644} C_VEL
LIN {X 0,Y 76.198,Z 646.951,A -85,B 0,C 180,E1 -27948.351,E2 -27948.351} C_VEL
LIN {X 0,Y 77.092,Z 647.591,A -85,B 0,C 180,E1 -27950.04,E2 -27950.04} C_VEL
LIN {X 0,Y 78.985,Z 650.828,A -85,B 0,C 180,E1 -27953.782,E2 -27953.782} C_VEL
LIN {X 0,Y 80.801,Z 652.607,A -85,B 0,C 180,E1 -27956.592,E2 -27956.592} C_VEL
LIN {X 0,Y 83.206,Z 656.253,A -85,B 0,C 180,E1 -27960.074,E2 -27960.074} C_VEL
LIN {X 0,Y 84.419,Z 657.708,A -85,B 0,C 180,E1 -27961.573,E2 -27961.573} C_VEL
LIN {X 0,Y 88.12,Z 663.334,A -85,B 0,C 180,E1 -27965.928,E2 -27965.928} C_VEL
LIN {X 0,Y 92.28,Z 669.827,A -85,B 0,C 180,E1 -27970.079,E2 -27970.079} C_VEL
LIN {X 0,Y 98.573,Z 681.69,A -85,B 0,C 180,E1 -27975.573,E2 -27975.573} C_VEL
LIN {X 0,Y 104.152,Z 695.976,A -85,B 0,C 180,E1 -27980.048,E2 -27980.048} C_VEL
LIN {X 0,Y 100.155,Z 732.389,A -85,B 0,C 180,E1 -27982.53,E2 -27982.53} C_VEL
LIN {X 0,Y 97.676,Z 746.331,A -85,B 0,C 180,E1 -27984.157,E2 -27984.157} C_VEL
LIN {X 0,Y 94.609,Z 758.616,A -85,B 0,C 180,E1 -27986.273,E2 -27986.273} C_VEL
LIN {X 0,Y 90.815,Z 770.793,A -85,B 0,C 180,E1 -27989.255,E2 -27989.255} C_VEL
LIN {X 0,Y 86.765,Z 781.752,A -85,B 0,C 180,E1 -27992.902,E2 -27992.902} C_VEL
LIN {X 0,Y 82.292,Z 792.529,A -85,B 0,C 180,E1 -27997.792,E2 -27997.792} C_VEL
LIN {X 0,Y 78.016,Z 802.27,A -85,B 0,C 180,E1 -28003.842,E2 -28003.842} C_VEL
LIN {X 0,Y 74.362,Z 810.803,A -85,B 0,C 180,E1 -28010.989,E2 -28010.989} C_VEL
LIN {X 0,Y 71.482,Z 818.264,A -85,B 0,C 180,E1 -28019.445,E2 -28019.445} C_VEL
LIN {X 0,Y 69.713,Z 824.509,A -85,B 0,C 180,E1 -28028.983,E2 -28028.983} C_VEL
LIN {X 0,Y 69.575,Z 829.461,A -85,B 0,C 180,E1 -28039.113,E2 -28039.113} C_VEL
LIN {X 0,Y 71.822,Z 833.518,A -85,B 0,C 180,E1 -28050.711,E2 -28050.711} C_VEL
LIN {X 0,Y 75.251,Z 835.526,A -85,B 0,C 180,E1 -28059.054,E2 -28059.054} C_VEL
LIN {X 0,Y 79.676,Z 836.543,A -85,B 0,C 180,E1 -28065.99,E2 -28065.99} C_VEL
LIN {X 0,Y 85.13,Z 836.755,A -85,B 0,C 180,E1 -28072.156,E2 -28072.156} C_VEL
LIN {X 0,Y 91.445,Z 836.158,A -85,B 0,C 180,E1 -28077.553,E2 -28077.553} C_VEL
LIN {X 0,Y 101.63,Z 833.954,A -85,B 0,C 180,E1 -28083.967,E2 -28083.967} C_VEL
LIN {X 0,Y 111.641,Z 830.529,A -85,B 0,C 180,E1 -28088.634,E2 -28088.634} C_VEL
LIN {X 0,Y 122.358,Z 825.609,A -85,B 0,C 180,E1 -28092.467,E2 -28092.467} C_VEL
LIN {X 0,Y 132.524,Z 819.657,A -85,B 0,C 180,E1 -28095.378,E2 -28095.378} C_VEL
LIN {X 0,Y 143.148,Z 811.965,A -85,B 0,C 180,E1 -28097.872,E2 -28097.872} C_VEL
LIN {X 0,Y 151.83,Z 804.342,A -85,B 0,C 180,E1 -28099.611,E2 -28099.611} C_VEL
LIN {X 0,Y 160.104,Z 795.653,A -85,B 0,C 180,E1 -28100.989,E2 -28100.989} C_VEL
LIN {X 0,Y 162.935,Z 792.252,A -85,B 0,C 180,E1 -28101.462,E2 -28101.462} C_VEL
LIN {X 0,Y 161.496,Z 794.09,A -85,B 0,C 180,E1 -28102.103,E2 -28102.103} C_VEL
LIN {X 0,Y 153.047,Z 803.528,A -85,B 0,C 180,E1 -28103.308,E2 -28103.308} C_VEL
LIN {X 0,Y 143.375,Z 812.458,A -85,B 0,C 180,E1 -28104.931,E2 -28104.931} C_VEL
LIN {X 0,Y 133.897,Z 819.755,A -85,B 0,C 180,E1 -28106.839,E2 -28106.839} C_VEL
LIN {X 0,Y 124.721,Z 825.737,A -85,B 0,C 180,E1 -28109.144,E2 -28109.144} C_VEL
LIN {X 0,Y 115.89,Z 830.596,A -85,B 0,C 180,E1 -28111.898,E2 -28111.898} C_VEL
LIN {X 0,Y 107.364,Z 834.465,A -85,B 0,C 180,E1 -28115.093,E2 -28115.093} C_VEL
LIN {X 0,Y 99.389,Z 837.424,A -85,B 0,C 180,E1 -28118.939,E2 -28118.939} C_VEL
LIN {X 0,Y 89.742,Z 840.042,A -85,B 0,C 180,E1 -28125.186,E2 -28125.186} C_VEL
LIN {X 0,Y 81.489,Z 841.26,A -85,B 0,C 180,E1 -28132.865,E2 -28132.865} C_VEL
LIN {X 0,Y 75.158,Z 841.101,A -85,B 0,C 180,E1 -28142.126,E2 -28142.126} C_VEL
LIN {X 0,Y 71.419,Z 839.504,A -85,B 0,C 180,E1 -28152.83,E2 -28152.83} C_VEL
LIN {X 0,Y 70.365,Z 836.459,A -85,B 0,C 180,E1 -28164.268,E2 -28164.268} C_VEL
LIN {X 0,Y 70.54,Z 834.29,A -85,B 0,C 180,E1 -28170,E2 -28170} C_VEL
LIN {X 0,Y 70.514,Z 829.862,A -85,B 0,C 180,E1 -28178.598,E2 -28178.598} C_VEL
LIN {X 0,Y 72.042,Z 823.018,A -85,B 0,C 180,E1 -28188.484,E2 -28188.484} C_VEL
LIN {X 0,Y 74.823,Z 815.542,A -85,B 0,C 180,E1 -28196.497,E2 -28196.497} C_VEL
LIN {X 0,Y 78.021,Z 807.854,A -85,B 0,C 180,E1 -28202.715,E2 -28202.715} C_VEL
LIN {X 0,Y 82.197,Z 798.569,A -85,B 0,C 180,E1 -28208.307,E2 -28208.307} C_VEL
LIN {X 0,Y 86.936,Z 787.318,A -85,B 0,C 180,E1 -28213.219,E2 -28213.219} C_VEL
LIN {X 0,Y 91.381,Z 775.39,A -85,B 0,C 180,E1 -28216.938,E2 -28216.938} C_VEL
LIN {X 0,Y 95.114,Z 763.178,A -85,B 0,C 180,E1 -28219.639,E2 -28219.639} C_VEL
LIN {X 0,Y 98.28,Z 750.001,A -85,B 0,C 180,E1 -28221.661,E2 -28221.661} C_VEL
LIN {X 0,Y 100.556,Z 735.816,A -85,B 0,C 180,E1 -28223.033,E2 -28223.033} C_VEL
LIN {X 0,Y 103.653,Z 705.754,A -85,B 0,C 180,E1 -28225.087,E2 -28225.087} C_VEL
LIN {X 0,Y 103.325,Z 701.644,A -85,B 0,C 180,E1 -28225.697,E2 -28225.697} C_VEL
LIN {X 0,Y 99.36,Z 687.896,A -85,B 0,C 180,E1 -28229.22,E2 -28229.22} C_VEL
LIN {X 0,Y 95.574,Z 676.946,A -85,B 0,C 180,E1 -28232.782,E2 -28232.782} C_VEL
LIN {X 0,Y 90.517,Z 667.494,A -85,B 0,C 180,E1 -28237.531,E2 -28237.531} C_VEL
LIN {X 0,Y 85.966,Z 660.113,A -85,B 0,C 180,E1 -28242.503,E2 -28242.503} C_VEL
LIN {X 0,Y 83.452,Z 656.207,A -85,B 0,C 180,E1 -28245.717,E2 -28245.717} C_VEL
LIN {X 0,Y 82.646,Z 655.267,A -85,B 0,C 180,E1 -28246.746,E2 -28246.746} C_VEL
LIN {X 0,Y 80.851,Z 653.99,A -85,B 0,C 180,E1 -28249.054,E2 -28249.054} C_VEL
LIN {X 0,Y 77.764,Z 653.37,A -85,B 0,C 180,E1 -28253.308,E2 -28253.308} C_VEL
LIN {X 0,Y 74.547,Z 652.788,A -85,B 0,C 180,E1 -28258.886,E2 -28258.886} C_VEL
LIN {X 0,Y 73.707,Z 652.095,A -85,B 0,C 180,E1 -28260.781,E2 -28260.781} C_VEL
LIN {X 0,Y 71.606,Z 649.021,A -85,B 0,C 180,E1 -28267.576,E2 -28267.576} C_VEL
LIN {X 0,Y 71.377,Z 648.294,A -85,B 0,C 180,E1 -28268.776,E2 -28268.776} C_VEL
LIN {X 0,Y 69.48,Z 647.938,A -85,B 0,C 180,E1 -28284.448,E2 -28284.448} C_VEL
LIN {X 0,Y 70.855,Z 648.447,A -85,B 0,C 180,E1 -28295.421,E2 -28295.421} C_VEL
LIN {X 0,Y 71.726,Z 651.039,A -85,B 0,C 180,E1 -28299.79,E2 -28299.79} C_VEL
LIN {X 0,Y 74.964,Z 654.213,A -85,B 0,C 180,E1 -28308.39,E2 -28308.39} C_VEL
LIN {X 0,Y 77.178,Z 657.693,A -85,B 0,C 180,E1 -28312.929,E2 -28312.929} C_VEL
LIN {X 0,Y 78.347,Z 659.099,A -85,B 0,C 180,E1 -28314.95,E2 -28314.95} C_VEL
LIN {X 0,Y 80.959,Z 662.801,A -85,B 0,C 180,E1 -28318.987,E2 -28318.987} C_VEL
LIN {X 0,Y 84.602,Z 668.536,A -85,B 0,C 180,E1 -28323.736,E2 -28323.736} C_VEL
LIN {X 0,Y 88.859,Z 675.604,A -85,B 0,C 180,E1 -28328.498,E2 -28328.498} C_VEL
LIN {X 0,Y 94.289,Z 686.48,A -85,B 0,C 180,E1 -28333.697,E2 -28333.697} C_VEL
LIN {X 0,Y 98.522,Z 697.85,A -85,B 0,C 180,E1 -28337.56,E2 -28337.56} C_VEL
LIN {X 0,Y 94.388,Z 733.759,A -85,B 0,C 180,E1 -28340.108,E2 -28340.108} C_VEL
LIN {X 0,Y 91.825,Z 747.015,A -85,B 0,C 180,E1 -28341.693,E2 -28341.693} C_VEL
LIN {X 0,Y 88.415,Z 759.843,A -85,B 0,C 180,E1 -28344.01,E2 -28344.01} C_VEL
LIN {X 0,Y 84.443,Z 771.738,A -85,B 0,C 180,E1 -28347.06,E2 -28347.06} C_VEL
LIN {X 0,Y 79.791,Z 783.501,A -85,B 0,C 180,E1 -28351.259,E2 -28351.259} C_VEL
LIN {X 0,Y 74.938,Z 794.378,A -85,B 0,C 180,E1 -28356.732,E2 -28356.732} C_VEL
LIN {X 0,Y 70.732,Z 803.314,A -85,B 0,C 180,E1 -28362.915,E2 -28362.915} C_VEL
LIN {X 0,Y 66.909,Z 811.858,A -85,B 0,C 180,E1 -28371.009,E2 -28371.009} C_VEL
LIN {X 0,Y 64.348,Z 818.26,A -85,B 0,C 180,E1 -28379.109,E2 -28379.109} C_VEL
LIN {X 0,Y 62.534,Z 824.786,A -85,B 0,C 180,E1 -28390.15,E2 -28390.15} C_VEL
LIN {X 0,Y 62.707,Z 829.86,A -85,B 0,C 180,E1 -28401.676,E2 -28401.676} C_VEL
LIN {X 0,Y 64.49,Z 832.874,A -85,B 0,C 180,E1 -28410.669,E2 -28410.669} C_VEL
LIN {X 0,Y 69.277,Z 835.745,A -85,B 0,C 180,E1 -28422.284,E2 -28422.284} C_VEL
LIN {X 0,Y 73.832,Z 836.787,A -85,B 0,C 180,E1 -28429.028,E2 -28429.028} C_VEL
LIN {X 0,Y 79.244,Z 837.159,A -85,B 0,C 180,E1 -28434.914,E2 -28434.914} C_VEL
LIN {X 0,Y 85.366,Z 836.898,A -85,B 0,C 180,E1 -28440.002,E2 -28440.002} C_VEL
LIN {X 0,Y 92.116,Z 835.927,A -85,B 0,C 180,E1 -28444.378,E2 -28444.378} C_VEL
LIN {X 0,Y 103.11,Z 833.249,A -85,B 0,C 180,E1 -28449.834,E2 -28449.834} C_VEL
LIN {X 0,Y 111.323,Z 830.349,A -85,B 0,C 180,E1 -28452.927,E2 -28452.927} C_VEL
LIN {X 0,Y 123.331,Z 824.852,A -85,B 0,C 180,E1 -28456.556,E2 -28456.556} C_VEL
LIN {X 0,Y 134.666,Z 818.136,A -85,B 0,C 180,E1 -28459.228,E2 -28459.228} C_VEL
LIN {X 0,Y 145.059,Z 810.442,A -85,B 0,C 180,E1 -28461.27,E2 -28461.27} C_VEL
LIN {X 0,Y 143.861,Z 811.496,A -85,B 0,C 180,E1 -28461.848,E2 -28461.848} C_VEL
LIN {X 0,Y 134.098,Z 818.909,A -85,B 0,C 180,E1 -28463.488,E2 -28463.488} C_VEL
LIN {X 0,Y 124.579,Z 824.953,A -85,B 0,C 180,E1 -28465.498,E2 -28465.498} C_VEL
LIN {X 0,Y 115.282,Z 829.868,A -85,B 0,C 180,E1 -28467.877,E2 -28467.877} C_VEL
LIN {X 0,Y 103.454,Z 834.884,A -85,B 0,C 180,E1 -28471.881,E2 -28471.881} C_VEL
LIN {X 0,Y 95.087,Z 837.602,A -85,B 0,C 180,E1 -28475.61,E2 -28475.61} C_VEL
LIN {X 0,Y 84.844,Z 839.966,A -85,B 0,C 180,E1 -28481.799,E2 -28481.799} C_VEL
LIN {X 0,Y 75.933,Z 840.939,A -85,B 0,C 180,E1 -28489.619,E2 -28489.619} C_VEL
LIN {X 0,Y 68.956,Z 840.496,A -85,B 0,C 180,E1 -28499.364,E2 -28499.364} C_VEL
LIN {X 0,Y 64.68,Z 838.697,A -85,B 0,C 180,E1 -28510.976,E2 -28510.976} C_VEL
LIN {X 0,Y 63.672,Z 837.263,A -85,B 0,C 180,E1 -28517.247,E2 -28517.247} C_VEL
LIN {X 0,Y 63.423,Z 834.664,A -85,B 0,C 180,E1 -28525.834,E2 -28525.834} C_VEL
LIN {X 0,Y 63.512,Z 833.091,A -85,B 0,C 180,E1 -28530,E2 -28530} C_VEL
LIN {X 0,Y 63.544,Z 828.45,A -85,B 0,C 180,E1 -28539.549,E2 -28539.549} C_VEL
LIN {X 0,Y 64.987,Z 822.487,A -85,B 0,C 180,E1 -28548.931,E2 -28548.931} C_VEL
LIN {X 0,Y 67.935,Z 814.978,A -85,B 0,C 180,E1 -28557.744,E2 -28557.744} C_VEL
LIN {X 0,Y 71.344,Z 807.243,A -85,B 0,C 180,E1 -28564.5,E2 -28564.5} C_VEL
LIN {X 0,Y 76.289,Z 796.828,A -85,B 0,C 180,E1 -28571.023,E2 -28571.023} C_VEL
LIN {X 0,Y 80.636,Z 787.017,A -85,B 0,C 180,E1 -28575.453,E2 -28575.453} C_VEL
LIN {X 0,Y 84.919,Z 776.163,A -85,B 0,C 180,E1 -28579.041,E2 -28579.041} C_VEL
LIN {X 0,Y 88.829,Z 764.297,A -85,B 0,C 180,E1 -28581.833,E2 -28581.833} C_VEL
LIN {X 0,Y 92.286,Z 750.915,A -85,B 0,C 180,E1 -28584.011,E2 -28584.011} C_VEL
LIN {X 0,Y 94.645,Z 737.954,A -85,B 0,C 180,E1 -28585.368,E2 -28585.368} C_VEL
LIN {X 0,Y 98.136,Z 706.363,A -85,B 0,C 180,E1 -28587.585,E2 -28587.585} C_VEL
LIN {X 0,Y 97.751,Z 703.36,A -85,B 0,C 180,E1 -28588.149,E2 -28588.149} C_VEL
LIN {X 0,Y 94.144,Z 690.25,A -85,B 0,C 180,E1 -28591.85,E2 -28591.85} C_VEL
LIN {X 0,Y 91.112,Z 680.981,A -85,B 0,C 180,E1 -28595.102,E2 -28595.102} C_VEL
LIN {X 0,Y 86.444,Z 672.039,A -85,B 0,C 180,E1 -28599.993,E2 -28599.993} C_VEL
LIN {X 0,Y 82.541,Z 665.37,A -85,B 0,C 180,E1 -28604.856,E2 -28604.856} C_VEL
LIN {X 0,Y 80.382,Z 661.918,A -85,B 0,C 180,E1 -28607.87,E2 -28607.87} C_VEL
LIN {X 0,Y 77.93,Z 657.938,A -85,B 0,C 180,E1 -28611.897,E2 -28611.897} C_VEL
LIN {X 0,Y 75.684,Z 654.504,A -85,B 0,C 180,E1 -28616.337,E2 -28616.337} C_VEL
LIN {X 0,Y 75.102,Z 653.448,A -85,B 0,C 180,E1 -28617.651,E2 -28617.651} C_VEL
LIN {X 0,Y 73.707,Z 652.095,A -85,B 0,C 180,E1 -28620.781,E2 -28620.781} C_VEL
LIN {X 0,Y 72.613,Z 651.21,A -85,B 0,C 180,E1 -28623.647,E2 -28623.647} C_VEL
LIN {X 0,Y 71.072,Z 651.17,A -85,B 0,C 180,E1 -28628.207,E2 -28628.207} C_VEL
LIN {X 0,Y 69.106,Z 653.026,A -85,B 0,C 180,E1 -28636.157,E2 -28636.157} C_VEL
LIN {X 0,Y 68.386,Z 654.886,A -85,B 0,C 180,E1 -28644.538,E2 -28644.538} C_VEL
LIN {X 0,Y 68.423,Z 655.004,A -85,B 0,C 180,E1 -28646.248,E2 -28646.248} C_VEL
LIN {X 0,Y 69.396,Z 655.458,A -85,B 0,C 180,E1 -28654.064,E2 -28654.064} C_VEL
LIN {X 0,Y 70.473,Z 658.235,A -85,B 0,C 180,E1 -28659.571,E2 -28659.571} C_VEL
LIN {X 0,Y 73.015,Z 660.946,A -85,B 0,C 180,E1 -28666.911,E2 -28666.911} C_VEL
LIN {X 0,Y 75.335,Z 664.47,A -85,B 0,C 180,E1 -28671.948,E2 -28671.948} C_VEL
LIN {X 0,Y 78.734,Z 669.827,A -85,B 0,C 180,E1 -28677.936,E2 -28677.936} C_VEL
LIN {X 0,Y 82.622,Z 676.123,A -85,B 0,C 180,E1 -28683.289,E2 -28683.289} C_VEL
LIN {X 0,Y 86.208,Z 682.984,A -85,B 0,C 180,E1 -28687.629,E2 -28687.629} C_VEL
LIN {X 0,Y 89.841,Z 690.735,A -85,B 0,C 180,E1 -28691.487,E2 -28691.487} C_VEL
LIN {X 0,Y 93.088,Z 699.737,A -85,B 0,C 180,E1 -28694.777,E2 -28694.777} C_VEL
LIN {X 0,Y 89.029,Z 733.496,A -85,B 0,C 180,E1 -28697.195,E2 -28697.195} C_VEL
LIN {X 0,Y 86.318,Z 747.043,A -85,B 0,C 180,E1 -28698.828,E2 -28698.828} C_VEL
LIN {X 0,Y 82.77,Z 759.78,A -85,B 0,C 180,E1 -28701.147,E2 -28701.147} C_VEL
LIN {X 0,Y 78.594,Z 771.598,A -85,B 0,C 180,E1 -28704.226,E2 -28704.226} C_VEL
LIN {X 0,Y 73.737,Z 783.239,A -85,B 0,C 180,E1 -28708.498,E2 -28708.498} C_VEL
LIN {X 0,Y 69.071,Z 793.176,A -85,B 0,C 180,E1 -28713.642,E2 -28713.642} C_VEL
LIN {X 0,Y 64.308,Z 802.627,A -85,B 0,C 180,E1 -28720.416,E2 -28720.416} C_VEL
LIN {X 0,Y 60.48,Z 810.58,A -85,B 0,C 180,E1 -28728.302,E2 -28728.302} C_VEL
LIN {X 0,Y 57.543,Z 817.309,A -85,B 0,C 180,E1 -28737.258,E2 -28737.258} C_VEL
LIN {X 0,Y 55.52,Z 823.995,A -85,B 0,C 180,E1 -28749.265,E2 -28749.265} C_VEL
LIN {X 0,Y 55.506,Z 828.755,A -85,B 0,C 180,E1 -28760.727,E2 -28760.727} C_VEL
LIN {X 0,Y 57.139,Z 832.027,A -85,B 0,C 180,E1 -28770.533,E2 -28770.533} C_VEL
LIN {X 0,Y 60.165,Z 834.452,A -85,B 0,C 180,E1 -28779.49,E2 -28779.49} C_VEL
LIN {X 0,Y 64.697,Z 836.254,A -85,B 0,C 180,E1 -28787.859,E2 -28787.859} C_VEL
LIN {X 0,Y 70.532,Z 837.313,A -85,B 0,C 180,E1 -28795.136,E2 -28795.136} C_VEL
LIN {X 0,Y 77.324,Z 837.558,A -85,B 0,C 180,E1 -28801.232,E2 -28801.232} C_VEL
LIN {X 0,Y 84.845,Z 837.034,A -85,B 0,C 180,E1 -28806.294,E2 -28806.294} C_VEL
LIN {X 0,Y 92.909,Z 835.748,A -85,B 0,C 180,E1 -28810.471,E2 -28810.471} C_VEL
LIN {X 0,Y 101.377,Z 833.689,A -85,B 0,C 180,E1 -28813.945,E2 -28813.945} C_VEL
LIN {X 0,Y 114.217,Z 829.155,A -85,B 0,C 180,E1 -28817.92,E2 -28817.92} C_VEL
LIN {X 0,Y 125.571,Z 823.757,A -85,B 0,C 180,E1 -28820.652,E2 -28820.652} C_VEL
LIN {X 0,Y 128.192,Z 822.279,A -85,B 0,C 180,E1 -28821.253,E2 -28821.253} C_VEL
LIN {X 0,Y 118.513,Z 827.626,A -85,B 0,C 180,E1 -28823.198,E2 -28823.198} C_VEL
LIN {X 0,Y 109.093,Z 831.912,A -85,B 0,C 180,E1 -28825.593,E2 -28825.593} C_VEL
LIN {X 0,Y 102.905,Z 834.247,A -85,B 0,C 180,E1 -28827.399,E2 -28827.399} C_VEL
LIN {X 0,Y 91.135,Z 837.78,A -85,B 0,C 180,E1 -28831.977,E2 -28831.977} C_VEL
LIN {X 0,Y 80.278,Z 839.846,A -85,B 0,C 180,E1 -28838.011,E2 -28838.011} C_VEL
LIN {X 0,Y 70.663,Z 840.535,A -85,B 0,C 180,E1 -28845.878,E2 -28845.878} C_VEL
LIN {X 0,Y 62.946,Z 839.875,A -85,B 0,C 180,E1 -28856.066,E2 -28856.066} C_VEL
LIN {X 0,Y 58.029,Z 837.836,A -85,B 0,C 180,E1 -28868.695,E2 -28868.695} C_VEL
LIN {X 0,Y 56.812,Z 836.269,A -85,B 0,C 180,E1 -28875.676,E2 -28875.676} C_VEL
LIN {X 0,Y 56.421,Z 833.562,A -85,B 0,C 180,E1 -28885.256,E2 -28885.256} C_VEL
LIN {X 0,Y 56.484,Z 831.856,A -85,B 0,C 180,E1 -28890,E2 -28890} C_VEL
LIN {X 0,Y 56.604,Z 826.971,A -85,B 0,C 180,E1 -28900.733,E2 -28900.733} C_VEL
LIN {X 0,Y 58.316,Z 820.727,A -85,B 0,C 180,E1 -28911.195,E2 -28911.195} C_VEL
LIN {X 0,Y 61.758,Z 812.865,A -85,B 0,C 180,E1 -28920.802,E2 -28920.802} C_VEL
LIN {X 0,Y 66.582,Z 803.032,A -85,B 0,C 180,E1 -28929.295,E2 -28929.295} C_VEL
LIN {X 0,Y 71.623,Z 792.8,A -85,B 0,C 180,E1 -28935.348,E2 -28935.348} C_VEL
LIN {X 0,Y 76.723,Z 781.521,A -85,B 0,C 180,E1 -28939.996,E2 -28939.996} C_VEL
LIN {X 0,Y 81.127,Z 770.198,A -85,B 0,C 180,E1 -28943.255,E2 -28943.255} C_VEL
LIN {X 0,Y 85.325,Z 756.46,A -85,B 0,C 180,E1 -28945.976,E2 -28945.976} C_VEL
LIN {X 0,Y 88.137,Z 743.965,A -85,B 0,C 180,E1 -28947.641,E2 -28947.641} C_VEL
LIN {X 0,Y 90.147,Z 730.22,A -85,B 0,C 180,E1 -28948.772,E2 -28948.772} C_VEL
LIN {X 0,Y 92.766,Z 706.598,A -85,B 0,C 180,E1 -28950.457,E2 -28950.457} C_VEL
LIN {X 0,Y 89.365,Z 693.507,A -85,B 0,C 180,E1 -28954.441,E2 -28954.441} C_VEL
LIN {X 0,Y 86.698,Z 684.994,A -85,B 0,C 180,E1 -28957.652,E2 -28957.652} C_VEL
LIN {X 0,Y 82.157,Z 675.773,A -85,B 0,C 180,E1 -28963.23,E2 -28963.23} C_VEL
LIN {X 0,Y 77.916,Z 668.233,A -85,B 0,C 180,E1 -28969.428,E2 -28969.428} C_VEL
LIN {X 0,Y 75.246,Z 663.808,A -85,B 0,C 180,E1 -28974.354,E2 -28974.354} C_VEL
LIN {X 0,Y 72.936,Z 659.838,A -85,B 0,C 180,E1 -28979.652,E2 -28979.652} C_VEL
LIN {X 0,Y 70.121,Z 655.817,A -85,B 0,C 180,E1 -28988.916,E2 -28988.916} C_VEL
LIN {X 0,Y 69.767,Z 655.195,A -85,B 0,C 180,E1 -28990.651,E2 -28990.651} C_VEL
LIN {X 0,Y 68.423,Z 655.004,A -85,B 0,C 180,E1 -29006.248,E2 -29006.248} C_VEL
LIN {X 0,Y 68.522,Z 655.725,A -85,B 0,C 180,E1 -29008.898,E2 -29008.898} C_VEL
LIN {X 0,Y 68.618,Z 658.147,A -85,B 0,C 180,E1 -29012.213,E2 -29012.213} C_VEL
LIN {X 0,Y 69.1,Z 664.299,A -85,B 0,C 180,E1 -29018.361,E2 -29018.361} C_VEL
LIN {X 0,Y 69.779,Z 666.042,A -85,B 0,C 180,E1 -29021.355,E2 -29021.355} C_VEL
LIN {X 0,Y 71.061,Z 667.564,A -85,B 0,C 180,E1 -29025.184,E2 -29025.184} C_VEL
LIN {X 0,Y 73.603,Z 671.732,A -85,B 0,C 180,E1 -29031.264,E2 -29031.264} C_VEL
LIN {X 0,Y 76.42,Z 676.53,A -85,B 0,C 180,E1 -29036.601,E2 -29036.601} C_VEL
LIN {X 0,Y 80.611,Z 683.969,A -85,B 0,C 180,E1 -29042.85,E2 -29042.85} C_VEL
LIN {X 0,Y 85.349,Z 694.441,A -85,B 0,C 180,E1 -29048.829,E2 -29048.829} C_VEL
LIN {X 0,Y 87.779,Z 701.864,A -85,B 0,C 180,E1 -29051.747,E2 -29051.747} C_VEL
LIN {X 0,Y 83.803,Z 733.436,A -85,B 0,C 180,E1 -29054.022,E2 -29054.022} C_VEL
LIN {X 0,Y 80.868,Z 747.391,A -85,B 0,C 180,E1 -29055.686,E2 -29055.686} C_VEL
LIN {X 0,Y 77.229,Z 759.848,A -85,B 0,C 180,E1 -29057.956,E2 -29057.956} C_VEL
LIN {X 0,Y 72.991,Z 771.287,A -85,B 0,C 180,E1 -29060.949,E2 -29060.949} C_VEL
LIN {X 0,Y 67.632,Z 783.475,A -85,B 0,C 180,E1 -29065.53,E2 -29065.53} C_VEL
LIN {X 0,Y 62.073,Z 794.456,A -85,B 0,C 180,E1 -29071.619,E2 -29071.619} C_VEL
LIN {X 0,Y 56.962,Z 803.973,A -85,B 0,C 180,E1 -29079.259,E2 -29079.259} C_VEL
LIN {X 0,Y 53.222,Z 811.189,A -85,B 0,C 180,E1 -29087.412,E2 -29087.412} C_VEL
LIN {X 0,Y 50.099,Z 817.985,A -85,B 0,C 180,E1 -29097.861,E2 -29097.861} C_VEL
LIN {X 0,Y 48.44,Z 823.454,A -85,B 0,C 180,E1 -29109.105,E2 -29109.105} C_VEL
LIN {X 0,Y 48.43,Z 827.953,A -85,B 0,C 180,E1 -29120.895,E2 -29120.895} C_VEL
LIN {X 0,Y 51.179,Z 832.512,A -85,B 0,C 180,E1 -29135.676,E2 -29135.676} C_VEL
LIN {X 0,Y 57.247,Z 835.766,A -85,B 0,C 180,E1 -29149.144,E2 -29149.144} C_VEL
LIN {X 0,Y 66.164,Z 837.613,A -85,B 0,C 180,E1 -29160.003,E2 -29160.003} C_VEL
LIN {X 0,Y 72.957,Z 837.963,A -85,B 0,C 180,E1 -29165.531,E2 -29165.531} C_VEL
LIN {X 0,Y 80.346,Z 837.696,A -85,B 0,C 180,E1 -29170.078,E2 -29170.078} C_VEL
LIN {X 0,Y 88.212,Z 836.72,A -85,B 0,C 180,E1 -29173.831,E2 -29173.831} C_VEL
LIN {X 0,Y 96.421,Z 835.102,A -85,B 0,C 180,E1 -29176.953,E2 -29176.953} C_VEL
LIN {X 0,Y 108.117,Z 831.675,A -85,B 0,C 180,E1 -29180.349,E2 -29180.349} C_VEL
LIN {X 0,Y 109.608,Z 831.156,A -85,B 0,C 180,E1 -29180.715,E2 -29180.715} C_VEL
LIN {X 0,Y 107.571,Z 831.996,A -85,B 0,C 180,E1 -29181.799,E2 -29181.799} C_VEL
LIN {X 0,Y 99.853,Z 834.7,A -85,B 0,C 180,E1 -29183.8,E2 -29183.8} C_VEL
LIN {X 0,Y 87.575,Z 837.875,A -85,B 0,C 180,E1 -29188.026,E2 -29188.026} C_VEL
LIN {X 0,Y 76.107,Z 839.673,A -85,B 0,C 180,E1 -29193.792,E2 -29193.792} C_VEL
LIN {X 0,Y 65.743,Z 840.125,A -85,B 0,C 180,E1 -29201.558,E2 -29201.558} C_VEL
LIN {X 0,Y 57.193,Z 839.188,A -85,B 0,C 180,E1 -29212.092,E2 -29212.092} C_VEL
LIN {X 0,Y 51.497,Z 836.885,A -85,B 0,C 180,E1 -29225.832,E2 -29225.832} C_VEL
LIN {X 0,Y 49.425,Z 833.138,A -85,B 0,C 180,E1 -29241.825,E2 -29241.825} C_VEL
LIN {X 0,Y 49.456,Z 830.553,A -85,B 0,C 180,E1 -29250,E2 -29250} C_VEL
LIN {X 0,Y 49.703,Z 825.418,A -85,B 0,C 180,E1 -29262.245,E2 -29262.245} C_VEL
LIN {X 0,Y 51.819,Z 818.854,A -85,B 0,C 180,E1 -29274.008,E2 -29274.008} C_VEL
LIN {X 0,Y 55.814,Z 810.668,A -85,B 0,C 180,E1 -29284.514,E2 -29284.514} C_VEL
LIN {X 0,Y 60.255,Z 802.225,A -85,B 0,C 180,E1 -29292.117,E2 -29292.117} C_VEL
LIN {X 0,Y 65.125,Z 793.046,A -85,B 0,C 180,E1 -29297.894,E2 -29297.894} C_VEL
LIN {X 0,Y 70.537,Z 781.74,A -85,B 0,C 180,E1 -29302.85,E2 -29302.85} C_VEL
LIN {X 0,Y 75.156,Z 770.682,A -85,B 0,C 180,E1 -29306.181,E2 -29306.181} C_VEL
LIN {X 0,Y 79.168,Z 758.722,A -85,B 0,C 180,E1 -29308.696,E2 -29308.696} C_VEL
LIN {X 0,Y 82.668,Z 744.539,A -85,B 0,C 180,E1 -29310.709,E2 -29310.709} C_VEL
LIN {X 0,Y 84.763,Z 731.412,A -85,B 0,C 180,E1 -29311.846,E2 -29311.846} C_VEL
LIN {X 0,Y 87.536,Z 708.321,A -85,B 0,C 180,E1 -29313.466,E2 -29313.466} C_VEL
LIN {X 0,Y 84.416,Z 695.62,A -85,B 0,C 180,E1 -29317.703,E2 -29317.703} C_VEL
LIN {X 0,Y 82.509,Z 689.054,A -85,B 0,C 180,E1 -29320.432,E2 -29320.432} C_VEL
LIN {X 0,Y 78.437,Z 680.339,A -85,B 0,C 180,E1 -29326.143,E2 -29326.143} C_VEL
LIN {X 0,Y 75,Z 673.812,A -85,B 0,C 180,E1 -29332.005,E2 -29332.005} C_VEL
LIN {X 0,Y 72.791,Z 669.789,A -85,B 0,C 180,E1 -29336.711,E2 -29336.711} C_VEL
LIN {X 0,Y 70.835,Z 666.193,A -85,B 0,C 180,E1 -29341.854,E2 -29341.854} C_VEL
LIN {X 0,Y 68.513,Z 662.219,A -85,B 0,C 180,E1 -29351.094,E2 -29351.094} C_VEL
LIN {X 0,Y 67.299,Z 662.011,A -85,B 0,C 180,E1 -29366.14,E2 -29366.14} C_VEL
LIN {X 0,Y 67.988,Z 662.392,A -85,B 0,C 180,E1 -29372.644,E2 -29372.644} C_VEL
LIN {X 0,Y 69.295,Z 665.491,A -85,B 0,C 180,E1 -29379.623,E2 -29379.623} C_VEL
LIN {X 0,Y 69.779,Z 666.042,A -85,B 0,C 180,E1 -29381.355,E2 -29381.355} C_VEL
LIN {X 0,Y 70.654,Z 667.512,A -85,B 0,C 180,E1 -29384.227,E2 -29384.227} C_VEL
LIN {X 0,Y 71.868,Z 670.915,A -85,B 0,C 180,E1 -29387.986,E2 -29387.986} C_VEL
LIN {X 0,Y 72.951,Z 675.161,A -85,B 0,C 180,E1 -29391.193,E2 -29391.193} C_VEL
LIN {X 0,Y 74.418,Z 681.528,A -85,B 0,C 180,E1 -29395.127,E2 -29395.127} C_VEL
LIN {X 0,Y 76.37,Z 687.611,A -85,B 0,C 180,E1 -29399.084,E2 -29399.084} C_VEL
LIN {X 0,Y 78.901,Z 693.18,A -85,B 0,C 180,E1 -29402.96,E2 -29402.96} C_VEL
LIN {X 0,Y 81.44,Z 699.534,A -85,B 0,C 180,E1 -29406.477,E2 -29406.477} C_VEL
LIN {X 0,Y 82.782,Z 704.006,A -85,B 0,C 180,E1 -29408.388,E2 -29408.388} C_VEL
LIN {X 0,Y 78.733,Z 733.982,A -85,B 0,C 180,E1 -29410.48,E2 -29410.48} C_VEL
LIN {X 0,Y 75.682,Z 747.796,A -85,B 0,C 180,E1 -29412.11,E2 -29412.11} C_VEL
LIN {X 0,Y 71.682,Z 760.654,A -85,B 0,C 180,E1 -29414.442,E2 -29414.442} C_VEL
LIN {X 0,Y 67.176,Z 772.111,A -85,B 0,C 180,E1 -29417.501,E2 -29417.501} C_VEL
LIN {X 0,Y 61.538,Z 784.073,A -85,B 0,C 180,E1 -29422.182,E2 -29422.182} C_VEL
LIN {X 0,Y 55.571,Z 794.976,A -85,B 0,C 180,E1 -29428.615,E2 -29428.615} C_VEL
LIN {X 0,Y 49.641,Z 805.149,A -85,B 0,C 180,E1 -29437.714,E2 -29437.714} C_VEL
LIN {X 0,Y 45.35,Z 812.854,A -85,B 0,C 180,E1 -29448.056,E2 -29448.056} C_VEL
LIN {X 0,Y 42.459,Z 819.108,A -85,B 0,C 180,E1 -29459.773,E2 -29459.773} C_VEL
LIN {X 0,Y 41.132,Z 824.443,A -85,B 0,C 180,E1 -29473.113,E2 -29473.113} C_VEL
LIN {X 0,Y 42.465,Z 829.77,A -85,B 0,C 180,E1 -29490.236,E2 -29490.236} C_VEL
LIN {X 0,Y 47.778,Z 834.121,A -85,B 0,C 180,E1 -29506.913,E2 -29506.913} C_VEL
LIN {X 0,Y 56.528,Z 836.999,A -85,B 0,C 180,E1 -29520.004,E2 -29520.004} C_VEL
LIN {X 0,Y 63.667,Z 838.048,A -85,B 0,C 180,E1 -29526.558,E2 -29526.558} C_VEL
LIN {X 0,Y 71.845,Z 838.368,A -85,B 0,C 180,E1 -29531.986,E2 -29531.986} C_VEL
LIN {X 0,Y 80.506,Z 837.952,A -85,B 0,C 180,E1 -29536.209,E2 -29536.209} C_VEL
LIN {X 0,Y 91.693,Z 836.373,A -85,B 0,C 180,E1 -29540.271,E2 -29540.271} C_VEL
LIN {X 0,Y 90.774,Z 836.681,A -85,B 0,C 180,E1 -29541.712,E2 -29541.712} C_VEL
LIN {X 0,Y 78.335,Z 838.892,A -85,B 0,C 180,E1 -29546.214,E2 -29546.214} C_VEL
LIN {X 0,Y 66.703,Z 839.709,A -85,B 0,C 180,E1 -29552.554,E2 -29552.554} C_VEL
LIN {X 0,Y 56.28,Z 839.193,A -85,B 0,C 180,E1 -29561.476,E2 -29561.476} C_VEL
LIN {X 0,Y 48.005,Z 837.348,A -85,B 0,C 180,E1 -29574.155,E2 -29574.155} C_VEL
LIN {X 0,Y 43.306,Z 834.096,A -85,B 0,C 180,E1 -29591.061,E2 -29591.061} C_VEL
LIN {X 0,Y 42.446,Z 830.733,A -85,B 0,C 180,E1 -29604.775,E2 -29604.775} C_VEL
LIN {X 0,Y 42.428,Z 829.128,A -85,B 0,C 180,E1 -29610,E2 -29610} C_VEL
LIN {X 0,Y 42.849,Z 823.743,A -85,B 0,C 180,E1 -29624.242,E2 -29624.242} C_VEL
LIN {X 0,Y 45.443,Z 816.911,A -85,B 0,C 180,E1 -29637.643,E2 -29637.643} C_VEL
LIN {X 0,Y 50.098,Z 808.303,A -85,B 0,C 180,E1 -29649.144,E2 -29649.144} C_VEL
LIN {X 0,Y 55.228,Z 799.471,A -85,B 0,C 180,E1 -29657.029,E2 -29657.029} C_VEL
LIN {X 0,Y 60.633,Z 789.827,A -85,B 0,C 180,E1 -29662.832,E2 -29662.832} C_VEL
LIN {X 0,Y 65.859,Z 779.296,A -85,B 0,C 180,E1 -29667.177,E2 -29667.177} C_VEL
LIN {X 0,Y 70.815,Z 767.416,A -85,B 0,C 180,E1 -29670.489,E2 -29670.489} C_VEL
LIN {X 0,Y 74.997,Z 754.745,A -85,B 0,C 180,E1 -29672.902,E2 -29672.902} C_VEL
LIN {X 0,Y 78.08,Z 741.896,A -85,B 0,C 180,E1 -29674.486,E2 -29674.486} C_VEL
LIN {X 0,Y 80.941,Z 722.612,A -85,B 0,C 180,E1 -29675.916,E2 -29675.916} C_VEL
LIN {X 0,Y 82.516,Z 709.813,A -85,B 0,C 180,E1 -29676.83,E2 -29676.83} C_VEL
LIN {X 0,Y 79.689,Z 697.419,A -85,B 0,C 180,E1 -29681.494,E2 -29681.494} C_VEL
LIN {X 0,Y 78.469,Z 693.074,A -85,B 0,C 180,E1 -29683.523,E2 -29683.523} C_VEL
LIN {X 0,Y 75.074,Z 685.292,A -85,B 0,C 180,E1 -29689.039,E2 -29689.039} C_VEL
LIN {X 0,Y 72.028,Z 678.955,A -85,B 0,C 180,E1 -29695.275,E2 -29695.275} C_VEL
LIN {X 0,Y 70.341,Z 675.584,A -85,B 0,C 180,E1 -29699.443,E2 -29699.443} C_VEL
LIN {X 0,Y 68.948,Z 672.623,A -85,B 0,C 180,E1 -29703.87,E2 -29703.87} C_VEL
LIN {X 0,Y 67.151,Z 669.227,A -85,B 0,C 180,E1 -29712.079,E2 -29712.079} C_VEL
LIN {X 0,Y 66.147,Z 668.995,A -85,B 0,C 180,E1 -29725.147,E2 -29725.147} C_VEL
LIN {X 0,Y 66.662,Z 669.394,A -85,B 0,C 180,E1 -29731.484,E2 -29731.484} C_VEL
LIN {X 0,Y 67.909,Z 672.418,A -85,B 0,C 180,E1 -29738.858,E2 -29738.858} C_VEL
LIN {X 0,Y 69.157,Z 674.011,A -85,B 0,C 180,E1 -29743.248,E2 -29743.248} C_VEL
LIN {X 0,Y 71.351,Z 678.08,A -85,B 0,C 180,E1 -29749.346,E2 -29749.346} C_VEL
LIN {X 0,Y 73.879,Z 682.695,A -85,B 0,C 180,E1 -29754.658,E2 -29754.658} C_VEL
LIN {X 0,Y 76.37,Z 687.611,A -85,B 0,C 180,E1 -29759.084,E2 -29759.084} C_VEL
LIN {X 0,Y 77.643,Z 691.822,A -85,B 0,C 180,E1 -29761.403,E2 -29761.403} C_VEL
LIN {X 0,Y 78.281,Z 696.723,A -85,B 0,C 180,E1 -29763.041,E2 -29763.041} C_VEL
LIN {X 0,Y 78.342,Z 702.024,A -85,B 0,C 180,E1 -29764.13,E2 -29764.13} C_VEL
LIN {X 0,Y 77.874,Z 707.455,A -85,B 0,C 180,E1 -29764.725,E2 -29764.725} C_VEL
LIN {X 0,Y 73.82,Z 735.082,A -85,B 0,C 180,E1 -29766.555,E2 -29766.555} C_VEL
LIN {X 0,Y 70.782,Z 748.116,A -85,B 0,C 180,E1 -29768.079,E2 -29768.079} C_VEL
LIN {X 0,Y 66.55,Z 760.975,A -85,B 0,C 180,E1 -29770.342,E2 -29770.342} C_VEL
LIN {X 0,Y 61.589,Z 772.734,A -85,B 0,C 180,E1 -29773.425,E2 -29773.425} C_VEL
LIN {X 0,Y 55.964,Z 783.986,A -85,B 0,C 180,E1 -29777.867,E2 -29777.867} C_VEL
LIN {X 0,Y 50.447,Z 793.48,A -85,B 0,C 180,E1 -29783.372,E2 -29783.372} C_VEL
LIN {X 0,Y 44.297,Z 803.203,A -85,B 0,C 180,E1 -29792.01,E2 -29792.01} C_VEL
LIN {X 0,Y 39.359,Z 811.143,A -85,B 0,C 180,E1 -29802.897,E2 -29802.897} C_VEL
LIN {X 0,Y 35.926,Z 817.494,A -85,B 0,C 180,E1 -29815.655,E2 -29815.655} C_VEL
LIN {X 0,Y 34.066,Z 824.219,A -85,B 0,C 180,E1 -29835.003,E2 -29835.003} C_VEL
LIN {X 0,Y 35.342,Z 828.631,A -85,B 0,C 180,E1 -29851.167,E2 -29851.167} C_VEL
LIN {X 0,Y 41.012,Z 833.378,A -85,B 0,C 180,E1 -29870.138,E2 -29870.138} C_VEL
LIN {X 0,Y 49.26,Z 836.4,A -85,B 0,C 180,E1 -29882.959,E2 -29882.959} C_VEL
LIN {X 0,Y 57.126,Z 837.935,A -85,B 0,C 180,E1 -29890.203,E2 -29890.203} C_VEL
LIN {X 0,Y 69.627,Z 838.774,A -85,B 0,C 180,E1 -29897.63,E2 -29897.63} C_VEL
LIN {X 0,Y 74.696,Z 838.688,A -85,B 0,C 180,E1 -29899.804,E2 -29899.804} C_VEL
LIN {X 0,Y 75.465,Z 838.735,A -85,B 0,C 180,E1 -29901.366,E2 -29901.366} C_VEL
LIN {X 0,Y 63.16,Z 839.3,A -85,B 0,C 180,E1 -29907.107,E2 -29907.107} C_VEL
LIN {X 0,Y 51.855,Z 838.544,A -85,B 0,C 180,E1 -29915.594,E2 -29915.594} C_VEL
LIN {X 0,Y 42.486,Z 836.397,A -85,B 0,C 180,E1 -29928.574,E2 -29928.574} C_VEL
LIN {X 0,Y 36.746,Z 832.887,A -85,B 0,C 180,E1 -29947.511,E2 -29947.511} C_VEL
LIN {X 0,Y 35.529,Z 829.338,A -85,B 0,C 180,E1 -29963.754,E2 -29963.754} C_VEL
LIN {X 0,Y 35.4,Z 827.668,A -85,B 0,C 180,E1 -29970,E2 -29970} C_VEL
LIN {X 0,Y 36.069,Z 821.981,A -85,B 0,C 180,E1 -29986.994,E2 -29986.994} C_VEL
LIN {X 0,Y 39.355,Z 814.775,A -85,B 0,C 180,E1 -30002.393,E2 -30002.393} C_VEL
LIN {X 0,Y 43.8,Z 807.4,A -85,B 0,C 180,E1 -30012.994,E2 -30012.994} C_VEL
LIN {X 0,Y 49.449,Z 798.492,A -85,B 0,C 180,E1 -30021.415,E2 -30021.415} C_VEL
LIN {X 0,Y 55.307,Z 788.781,A -85,B 0,C 180,E1 -30027.334,E2 -30027.334} C_VEL
LIN {X 0,Y 60.882,Z 778.076,A -85,B 0,C 180,E1 -30031.664,E2 -30031.664} C_VEL
LIN {X 0,Y 66.038,Z 766.322,A -85,B 0,C 180,E1 -30034.802,E2 -30034.802} C_VEL
LIN {X 0,Y 70.151,Z 754.379,A -85,B 0,C 180,E1 -30036.986,E2 -30036.986} C_VEL
LIN {X 0,Y 73.48,Z 741.068,A -85,B 0,C 180,E1 -30038.545,E2 -30038.545} C_VEL
LIN {X 0,Y 76.451,Z 721.731,A -85,B 0,C 180,E1 -30039.907,E2 -30039.907} C_VEL
LIN {X 0,Y 77.728,Z 711.15,A -85,B 0,C 180,E1 -30040.733,E2 -30040.733} C_VEL
LIN {X 0,Y 75.18,Z 698.85,A -85,B 0,C 180,E1 -30045.822,E2 -30045.822} C_VEL
LIN {X 0,Y 72.333,Z 691.188,A -85,B 0,C 180,E1 -30051.325,E2 -30051.325} C_VEL
LIN {X 0,Y 69.595,Z 684.857,A -85,B 0,C 180,E1 -30057.754,E2 -30057.754} C_VEL
LIN {X 0,Y 68.044,Z 681.329,A -85,B 0,C 180,E1 -30062.432,E2 -30062.432} C_VEL
LIN {X 0,Y 67.058,Z 678.862,A -85,B 0,C 180,E1 -30066.399,E2 -30066.399} C_VEL
LIN {X 0,Y 65.751,Z 676.118,A -85,B 0,C 180,E1 -30073.53,E2 -30073.53} C_VEL
LIN {X 0,Y 65.351,Z 676.17,A -85,B 0,C 180,E1 -30089.889,E2 -30089.889} C_VEL
LIN {X 0,Y 66.535,Z 679.35,A -85,B 0,C 180,E1 -30098.104,E2 -30098.104} C_VEL
LIN {X 0,Y 67.456,Z 680.806,A -85,B 0,C 180,E1 -30101.723,E2 -30101.723} C_VEL
LIN {X 0,Y 69.167,Z 684.387,A -85,B 0,C 180,E1 -30107.264,E2 -30107.264} C_VEL
LIN {X 0,Y 71.612,Z 689.272,A -85,B 0,C 180,E1 -30113.036,E2 -30113.036} C_VEL
LIN {X 0,Y 74.484,Z 695.781,A -85,B 0,C 180,E1 -30118.672,E2 -30118.672} C_VEL
LIN {X 0,Y 77.322,Z 703.515,A -85,B 0,C 180,E1 -30123.432,E2 -30123.432} C_VEL
LIN {X 0,Y 78.047,Z 706.224,A -85,B 0,C 180,E1 -30124.653,E2 -30124.653} C_VEL
LIN {X 0,Y 77.874,Z 707.455,A -85,B 0,C 180,E1 -30124.725,E2 -30124.725} C_VEL
LIN {X 0,Y 76.724,Z 713.24,A -85,B 0,C 180,E1 -30124.725,E2 -30124.725} C_VEL
LIN {X 0,Y 71.16,Z 729.975,A -85,B 0,C 180,E1 -30122.553,E2 -30122.553} C_VEL
LIN {X 0,Y 69.458,Z 735.646,A -85,B 0,C 180,E1 -30122.201,E2 -30122.201} C_VEL
LIN {X 0,Y 68.982,Z 737.566,A -85,B 0,C 180,E1 -30122.279,E2 -30122.279} C_VEL
LIN {X 0,Y 65.687,Z 750.256,A -85,B 0,C 180,E1 -30123.739,E2 -30123.739} C_VEL
LIN {X 0,Y 61.201,Z 762.76,A -85,B 0,C 180,E1 -30125.916,E2 -30125.916} C_VEL
LIN {X 0,Y 56.075,Z 774.076,A -85,B 0,C 180,E1 -30128.85,E2 -30128.85} C_VEL
LIN {X 0,Y 49.652,Z 785.786,A -85,B 0,C 180,E1 -30133.556,E2 -30133.556} C_VEL
LIN {X 0,Y 42.746,Z 796.529,A -85,B 0,C 180,E1 -30140.537,E2 -30140.537} C_VEL
LIN {X 0,Y 36.51,Z 805.402,A -85,B 0,C 180,E1 -30150,E2 -30150} C_VEL
LIN {X 0,Y 31.369,Z 812.874,A -85,B 0,C 180,E1 -30162.946,E2 -30162.946} C_VEL
LIN {X 0,Y 27.944,Z 819.253,A -85,B 0,C 180,E1 -30180.198,E2 -30180.198} C_VEL
LIN {X 0,Y 27.466,Z 825.742,A -85,B 0,C 180,E1 -30205.388,E2 -30205.388} C_VEL
LIN {X 0,Y 31.54,Z 830.66,A -85,B 0,C 180,E1 -30227.131,E2 -30227.131} C_VEL
LIN {X 0,Y 37.254,Z 833.761,A -85,B 0,C 180,E1 -30240.006,E2 -30240.006} C_VEL
LIN {X 0,Y 44.26,Z 836.085,A -85,B 0,C 180,E1 -30249.141,E2 -30249.141} C_VEL
LIN {X 0,Y 52.145,Z 837.78,A -85,B 0,C 180,E1 -30255.642,E2 -30255.642} C_VEL
LIN {X 0,Y 60.517,Z 838.809,A -85,B 0,C 180,E1 -30260.393,E2 -30260.393} C_VEL
LIN {X 0,Y 60.253,Z 838.829,A -85,B 0,C 180,E1 -30261.076,E2 -30261.076} C_VEL
LIN {X 0,Y 48.084,Z 837.77,A -85,B 0,C 180,E1 -30268.724,E2 -30268.724} C_VEL
LIN {X 0,Y 37.487,Z 835.402,A -85,B 0,C 180,E1 -30281.418,E2 -30281.418} C_VEL
LIN {X 0,Y 30.38,Z 831.623,A -85,B 0,C 180,E1 -30302.442,E2 -30302.442} C_VEL
LIN {X 0,Y 28.595,Z 827.72,A -85,B 0,C 180,E1 -30322.934,E2 -30322.934} C_VEL
LIN {X 0,Y 28.352,Z 824.165,A -85,B 0,C 180,E1 -30337.401,E2 -30337.401} C_VEL
LIN {X 0,Y 30.471,Z 817.787,A -85,B 0,C 180,E1 -30357.469,E2 -30357.469} C_VEL
LIN {X 0,Y 35.623,Z 809.689,A -85,B 0,C 180,E1 -30373.669,E2 -30373.669} C_VEL
LIN {X 0,Y 41.414,Z 801.324,A -85,B 0,C 180,E1 -30383.712,E2 -30383.712} C_VEL
LIN {X 0,Y 48.233,Z 791.11,A -85,B 0,C 180,E1 -30390.954,E2 -30390.954} C_VEL
LIN {X 0,Y 54.841,Z 779.694,A -85,B 0,C 180,E1 -30395.933,E2 -30395.933} C_VEL
LIN {X 0,Y 60.224,Z 768.519,A -85,B 0,C 180,E1 -30398.997,E2 -30398.997} C_VEL
LIN {X 0,Y 65.142,Z 755.462,A -85,B 0,C 180,E1 -30401.335,E2 -30401.335} C_VEL
LIN {X 0,Y 68.614,Z 742.886,A -85,B 0,C 180,E1 -30402.817,E2 -30402.817} C_VEL
LIN {X 0,Y 71.177,Z 728.3,A -85,B 0,C 180,E1 -30403.86,E2 -30403.86} C_VEL
LIN {X 0,Y 73.277,Z 712.974,A -85,B 0,C 180,E1 -30404.874,E2 -30404.874} C_VEL
LIN {X 0,Y 71.406,Z 702.338,A -85,B 0,C 180,E1 -30409.731,E2 -30409.731} C_VEL
LIN {X 0,Y 69.214,Z 695.931,A -85,B 0,C 180,E1 -30414.945,E2 -30414.945} C_VEL
LIN {X 0,Y 67.151,Z 690.442,A -85,B 0,C 180,E1 -30420.876,E2 -30420.876} C_VEL
LIN {X 0,Y 65.933,Z 686.984,A -85,B 0,C 180,E1 -30425.701,E2 -30425.701} C_VEL
LIN {X 0,Y 65.237,Z 685.008,A -85,B 0,C 180,E1 -30429.331,E2 -30429.331} C_VEL
LIN {X 0,Y 64.435,Z 683.063,A -85,B 0,C 180,E1 -30434.711,E2 -30434.711} C_VEL
LIN {X 0,Y 64.098,Z 683.179,A -85,B 0,C 180,E1 -30448.702,E2 -30448.702} C_VEL
LIN {X 0,Y 65.435,Z 686.653,A -85,B 0,C 180,E1 -30458.45,E2 -30458.45} C_VEL
LIN {X 0,Y 66.981,Z 690.401,A -85,B 0,C 180,E1 -30464.692,E2 -30464.692} C_VEL
LIN {X 0,Y 69.07,Z 695.29,A -85,B 0,C 180,E1 -30470.664,E2 -30470.664} C_VEL
LIN {X 0,Y 71.305,Z 701.016,A -85,B 0,C 180,E1 -30475.753,E2 -30475.753} C_VEL
LIN {X 0,Y 73.456,Z 707.626,A -85,B 0,C 180,E1 -30480.142,E2 -30480.142} C_VEL
LIN {X 0,Y 73.558,Z 708.43,A -85,B 0,C 180,E1 -30480.44,E2 -30480.44} C_VEL
LIN {X 0,Y 69.384,Z 735.567,A -85,B 0,C 180,E1 -30482.102,E2 -30482.102} C_VEL
LIN {X 0,Y 68.982,Z 737.566,A -85,B 0,C 180,E1 -30482.279,E2 -30482.279} C_VEL
LIN {X 0,Y 67.225,Z 743.219,A -85,B 0,C 180,E1 -30482.261,E2 -30482.261} C_VEL
LIN {X 0,Y 62.988,Z 752.127,A -85,B 0,C 180,E1 -30481.301,E2 -30481.301} C_VEL
LIN {X 0,Y 58.201,Z 760.796,A -85,B 0,C 180,E1 -30480.534,E2 -30480.534} C_VEL
LIN {X 0,Y 55.554,Z 766.077,A -85,B 0,C 180,E1 -30481.044,E2 -30481.044} C_VEL
LIN {X 0,Y 50.023,Z 776.969,A -85,B 0,C 180,E1 -30483.846,E2 -30483.846} C_VEL
LIN {X 0,Y 43.231,Z 788.097,A -85,B 0,C 180,E1 -30488.426,E2 -30488.426} C_VEL
LIN {X 0,Y 36.406,Z 797.635,A -85,B 0,C 180,E1 -30494.823,E2 -30494.823} C_VEL
LIN {X 0,Y 29.312,Z 806.725,A -85,B 0,C 180,E1 -30505.734,E2 -30505.734} C_VEL
LIN {X 0,Y 23.392,Z 814.47,A -85,B 0,C 180,E1 -30523.022,E2 -30523.022} C_VEL
LIN {X 0,Y 20.185,Z 820.751,A -85,B 0,C 180,E1 -30547.533,E2 -30547.533} C_VEL
LIN {X 0,Y 22.206,Z 827.166,A -85,B 0,C 180,E1 -30581.704,E2 -30581.704} C_VEL
LIN {X 0,Y 31.325,Z 832.769,A -85,B 0,C 180,E1 -30606.894,E2 -30606.894} C_VEL
LIN {X 0,Y 42.915,Z 836.458,A -85,B 0,C 180,E1 -30619.124,E2 -30619.124} C_VEL
LIN {X 0,Y 45.115,Z 836.991,A -85,B 0,C 180,E1 -30620.829,E2 -30620.829} C_VEL
LIN {X 0,Y 33.255,Z 834.304,A -85,B 0,C 180,E1 -30632.292,E2 -30632.292} C_VEL
LIN {X 0,Y 24.411,Z 830.265,A -85,B 0,C 180,E1 -30654.845,E2 -30654.845} C_VEL
LIN {X 0,Y 21.735,Z 826.121,A -85,B 0,C 180,E1 -30680.687,E2 -30680.687} C_VEL
LIN {X 0,Y 21.439,Z 822.271,A -85,B 0,C 180,E1 -30700.387,E2 -30700.387} C_VEL
LIN {X 0,Y 24.461,Z 815.68,A -85,B 0,C 180,E1 -30725.072,E2 -30725.072} C_VEL
LIN {X 0,Y 30.919,Z 807.131,A -85,B 0,C 180,E1 -30742.705,E2 -30742.705} C_VEL
LIN {X 0,Y 37.691,Z 798.342,A -85,B 0,C 180,E1 -30752.335,E2 -30752.335} C_VEL
LIN {X 0,Y 44.458,Z 788.791,A -85,B 0,C 180,E1 -30758.234,E2 -30758.234} C_VEL
LIN {X 0,Y 50.772,Z 778.398,A -85,B 0,C 180,E1 -30762.107,E2 -30762.107} C_VEL
LIN {X 0,Y 56.443,Z 766.914,A -85,B 0,C 180,E1 -30764.788,E2 -30764.788} C_VEL
LIN {X 0,Y 61.146,Z 754.83,A -85,B 0,C 180,E1 -30766.612,E2 -30766.612} C_VEL
LIN {X 0,Y 64.69,Z 742.374,A -85,B 0,C 180,E1 -30767.888,E2 -30767.888} C_VEL
LIN {X 0,Y 67.183,Z 728.849,A -85,B 0,C 180,E1 -30768.736,E2 -30768.736} C_VEL
LIN {X 0,Y 69.208,Z 714.549,A -85,B 0,C 180,E1 -30769.641,E2 -30769.641} C_VEL
LIN {X 0,Y 68.025,Z 706.35,A -85,B 0,C 180,E1 -30773.81,E2 -30773.81} C_VEL
LIN {X 0,Y 66.257,Z 700.384,A -85,B 0,C 180,E1 -30779.059,E2 -30779.059} C_VEL
LIN {X 0,Y 64.727,Z 695.272,A -85,B 0,C 180,E1 -30785.174,E2 -30785.174} C_VEL
LIN {X 0,Y 63.768,Z 691.748,A -85,B 0,C 180,E1 -30790.828,E2 -30790.828} C_VEL
LIN {X 0,Y 63.174,Z 690.027,A -85,B 0,C 180,E1 -30795.705,E2 -30795.705} C_VEL
LIN {X 0,Y 62.883,Z 690.239,A -85,B 0,C 180,E1 -30807.692,E2 -30807.692} C_VEL
LIN {X 0,Y 63.996,Z 693.769,A -85,B 0,C 180,E1 -30817.521,E2 -30817.521} C_VEL
LIN {X 0,Y 65.098,Z 696.946,A -85,B 0,C 180,E1 -30822.679,E2 -30822.679} C_VEL
LIN {X 0,Y 66.566,Z 701.043,A -85,B 0,C 180,E1 -30827.841,E2 -30827.841} C_VEL
LIN {X 0,Y 68.26,Z 706.112,A -85,B 0,C 180,E1 -30832.559,E2 -30832.559} C_VEL
LIN {X 0,Y 69.546,Z 710.424,A -85,B 0,C 180,E1 -30835.706,E2 -30835.706} C_VEL
LIN {X 0,Y 65.399,Z 736.2,A -85,B 0,C 180,E1 -30837.112,E2 -30837.112} C_VEL
LIN {X 0,Y 61.818,Z 749.828,A -85,B 0,C 180,E1 -30838.408,E2 -30838.408} C_VEL
LIN {X 0,Y 56.923,Z 762.931,A -85,B 0,C 180,E1 -30840.406,E2 -30840.406} C_VEL
LIN {X 0,Y 55.554,Z 766.077,A -85,B 0,C 180,E1 -30841.044,E2 -30841.044} C_VEL
LIN {X 0,Y 52.701,Z 771.238,A -85,B 0,C 180,E1 -30841.597,E2 -30841.597} C_VEL
LIN {X 0,Y 46.712,Z 779.159,A -85,B 0,C 180,E1 -30840.965,E2 -30840.965} C_VEL
LIN {X 0,Y 40.205,Z 786.694,A -85,B 0,C 180,E1 -30840.537,E2 -30840.537} C_VEL
LIN {X 0,Y 36.536,Z 791.253,A -85,B 0,C 180,E1 -30841.98,E2 -30841.98} C_VEL
LIN {X 0,Y 28.079,Z 801.644,A -85,B 0,C 180,E1 -30849.658,E2 -30849.658} C_VEL
LIN {X 0,Y 20.092,Z 810.429,A -85,B 0,C 180,E1 -30863.853,E2 -30863.853} C_VEL
LIN {X 0,Y 14.707,Z 816.809,A -85,B 0,C 180,E1 -30887.155,E2 -30887.155} C_VEL
LIN {X 0,Y 14.022,Z 823.975,A -85,B 0,C 180,E1 -30937.447,E2 -30937.447} C_VEL
LIN {X 0,Y 21.34,Z 829.443,A -85,B 0,C 180,E1 -30968.894,E2 -30968.894} C_VEL
LIN {X 0,Y 28.351,Z 832.535,A -85,B 0,C 180,E1 -30979.429,E2 -30979.429} C_VEL
LIN {X 0,Y 24.175,Z 831.176,A -85,B 0,C 180,E1 -30989.296,E2 -30989.296} C_VEL
LIN {X 0,Y 15.797,Z 826.048,A -85,B 0,C 180,E1 -31023.584,E2 -31023.584} C_VEL
LIN {X 0,Y 14.965,Z 824.573,A -85,B 0,C 180,E1 -31035.633,E2 -31035.633} C_VEL
LIN {X 0,Y 14.704,Z 820.108,A -85,B 0,C 180,E1 -31067.03,E2 -31067.03} C_VEL
LIN {X 0,Y 20.341,Z 812.089,A -85,B 0,C 180,E1 -31101.02,E2 -31101.02} C_VEL
LIN {X 0,Y 27.212,Z 804.441,A -85,B 0,C 180,E1 -31114.676,E2 -31114.676} C_VEL
LIN {X 0,Y 35.812,Z 794.126,A -85,B 0,C 180,E1 -31123.076,E2 -31123.076} C_VEL
LIN {X 0,Y 43.212,Z 783.732,A -85,B 0,C 180,E1 -31127.375,E2 -31127.375} C_VEL
LIN {X 0,Y 49.929,Z 772.124,A -85,B 0,C 180,E1 -31130.161,E2 -31130.161} C_VEL
LIN {X 0,Y 55.881,Z 758.988,A -85,B 0,C 180,E1 -31132.051,E2 -31132.051} C_VEL
LIN {X 0,Y 60.207,Z 745.889,A -85,B 0,C 180,E1 -31133.238,E2 -31133.238} C_VEL
LIN {X 0,Y 63.211,Z 732.26,A -85,B 0,C 180,E1 -31134.013,E2 -31134.013} C_VEL
LIN {X 0,Y 65.636,Z 716.336,A -85,B 0,C 180,E1 -31134.819,E2 -31134.819} C_VEL
LIN {X 0,Y 64.964,Z 710.518,A -85,B 0,C 180,E1 -31138.071,E2 -31138.071} C_VEL
LIN {X 0,Y 63.725,Z 705.093,A -85,B 0,C 180,E1 -31143.264,E2 -31143.264} C_VEL
LIN {X 0,Y 62.577,Z 699.924,A -85,B 0,C 180,E1 -31150.174,E2 -31150.174} C_VEL
LIN {X 0,Y 62.198,Z 698.149,A -85,B 0,C 180,E1 -31153.453,E2 -31153.453} C_VEL
LIN {X 0,Y 61.923,Z 697.021,A -85,B 0,C 180,E1 -31156.741,E2 -31156.741} C_VEL
LIN {X 0,Y 61.688,Z 697.208,A -85,B 0,C 180,E1 -31166.506,E2 -31166.506} C_VEL
LIN {X 0,Y 62.429,Z 700.458,A -85,B 0,C 180,E1 -31175.668,E2 -31175.668} C_VEL
LIN {X 0,Y 63.606,Z 704.497,A -85,B 0,C 180,E1 -31182.039,E2 -31182.039} C_VEL
LIN {X 0,Y 65.232,Z 710.425,A -85,B 0,C 180,E1 -31188.456,E2 -31188.456} C_VEL
LIN {X 0,Y 65.842,Z 713.055,A -85,B 0,C 180,E1 -31190.531,E2 -31190.531} C_VEL
LIN {X 0,Y 61.881,Z 736.542,A -85,B 0,C 180,E1 -31191.546,E2 -31191.546} C_VEL
LIN {X 0,Y 58.301,Z 749.754,A -85,B 0,C 180,E1 -31192.526,E2 -31192.526} C_VEL
LIN {X 0,Y 53.118,Z 763.204,A -85,B 0,C 180,E1 -31194.149,E2 -31194.149} C_VEL
LIN {X 0,Y 47.368,Z 774.624,A -85,B 0,C 180,E1 -31196.195,E2 -31196.195} C_VEL
LIN {X 0,Y 40.223,Z 786.152,A -85,B 0,C 180,E1 -31199.698,E2 -31199.698} C_VEL
LIN {X 0,Y 36.536,Z 791.253,A -85,B 0,C 180,E1 -31201.98,E2 -31201.98} C_VEL
LIN {X 0,Y 32.761,Z 795.689,A -85,B 0,C 180,E1 -31203.833,E2 -31203.833} C_VEL
LIN {X 0,Y 25.35,Z 802.227,A -85,B 0,C 180,E1 -31204.626,E2 -31204.626} C_VEL
LIN {X 0,Y 17.403,Z 808.289,A -85,B 0,C 180,E1 -31206.042,E2 -31206.042} C_VEL
LIN {X 0,Y 12.902,Z 811.89,A -85,B 0,C 180,E1 -31211.969,E2 -31211.969} C_VEL
LIN {X 0,Y 6.257,Z 818.646,A -85,B 0,C 180,E1 -31258.352,E2 -31258.352} C_VEL
LIN {X 0,Y 10.152,Z 824.42,A -85,B 0,C 180,E1 -31329.987,E2 -31329.987} C_VEL
LIN {X 0,Y 14.302,Z 826.778,A -85,B 0,C 180,E1 -31341.641,E2 -31341.641} C_VEL
LIN {X 0,Y 10.077,Z 824.356,A -85,B 0,C 180,E1 -31365.78,E2 -31365.78} C_VEL
LIN {X 0,Y 7.896,Z 822.019,A -85,B 0,C 180,E1 -31392.835,E2 -31392.835} C_VEL
LIN {X 0,Y 9.783,Z 816.238,A -85,B 0,C 180,E1 -31455.919,E2 -31455.919} C_VEL
LIN {X 0,Y 18.445,Z 808.163,A -85,B 0,C 180,E1 -31482.278,E2 -31482.278} C_VEL
LIN {X 0,Y 26.716,Z 799.784,A -85,B 0,C 180,E1 -31490.56,E2 -31490.56} C_VEL
LIN {X 0,Y 35.3,Z 789.59,A -85,B 0,C 180,E1 -31494.521,E2 -31494.521} C_VEL
LIN {X 0,Y 43.108,Z 778.138,A -85,B 0,C 180,E1 -31496.918,E2 -31496.918} C_VEL
LIN {X 0,Y 49.22,Z 766.879,A -85,B 0,C 180,E1 -31498.173,E2 -31498.173} C_VEL
LIN {X 0,Y 54.473,Z 754.388,A -85,B 0,C 180,E1 -31499.047,E2 -31499.047} C_VEL
LIN {X 0,Y 58.434,Z 741.281,A -85,B 0,C 180,E1 -31499.717,E2 -31499.717} C_VEL
LIN {X 0,Y 61.079,Z 727.5,A -85,B 0,C 180,E1 -31500.202,E2 -31500.202} C_VEL
LIN {X 0,Y 62.538,Z 717.995,A -85,B 0,C 180,E1 -31500.625,E2 -31500.625} C_VEL
LIN {X 0,Y 62.295,Z 714.604,A -85,B 0,C 180,E1 -31502.766,E2 -31502.766} C_VEL
LIN {X 0,Y 61.388,Z 708.848,A -85,B 0,C 180,E1 -31509.025,E2 -31509.025} C_VEL
LIN {X 0,Y 60.837,Z 704.847,A -85,B 0,C 180,E1 -31515.243,E2 -31515.243} C_VEL
LIN {X 0,Y 60.632,Z 704.007,A -85,B 0,C 180,E1 -31518.568,E2 -31518.568} C_VEL
LIN {X 0,Y 60.524,Z 704.14,A -85,B 0,C 180,E1 -31525.232,E2 -31525.232} C_VEL
LIN {X 0,Y 60.915,Z 707.038,A -85,B 0,C 180,E1 -31533.535,E2 -31533.535} C_VEL
LIN {X 0,Y 61.93,Z 711.771,A -85,B 0,C 180,E1 -31540.639,E2 -31540.639} C_VEL
LIN {X 0,Y 62.682,Z 715.596,A -85,B 0,C 180,E1 -31544.67,E2 -31544.67} C_VEL
LIN {X 0,Y 59.202,Z 736.055,A -85,B 0,C 180,E1 -31545.344,E2 -31545.344} C_VEL
LIN {X 0,Y 55.409,Z 749.887,A -85,B 0,C 180,E1 -31545.995,E2 -31545.995} C_VEL
LIN {X 0,Y 50.555,Z 762.315,A -85,B 0,C 180,E1 -31546.863,E2 -31546.863} C_VEL
LIN {X 0,Y 44.18,Z 774.723,A -85,B 0,C 180,E1 -31548.219,E2 -31548.219} C_VEL
LIN {X 0,Y 37.115,Z 785.689,A -85,B 0,C 180,E1 -31550.274,E2 -31550.274} C_VEL
LIN {X 0,Y 28.474,Z 796.49,A -85,B 0,C 180,E1 -31553.873,E2 -31553.873} C_VEL
LIN {X 0,Y 18.665,Z 806.678,A -85,B 0,C 180,E1 -31561.923,E2 -31561.923} C_VEL
LIN {X 0,Y 12.902,Z 811.89,A -85,B 0,C 180,E1 -31571.969,E2 -31571.969} C_VEL
LIN {X 0,Y 11.781,Z 812.392,A -85,B 0,C 180,E1 -31570.87,E2 -31570.87} C_VEL
LIN {X 0,Y 10.341,Z 812.306,A -85,B 0,C 180,E1 -31560.69,E2 -31560.69} C_VEL
LIN {X 0,Y 10.53,Z 810.915,A -85,B 0,C 180,E1 -31537.707,E2 -31537.707} C_VEL
LIN {X 0,Y 12.209,Z 809.267,A -85,B 0,C 180,E1 -31525.054,E2 -31525.054} C_VEL
LIN {X 0,Y 15.925,Z 806.202,A -85,B 0,C 180,E1 -31514.345,E2 -31514.345} C_VEL
LIN {X 0,Y 21.937,Z 801.073,A -85,B 0,C 180,E1 -31507.274,E2 -31507.274} C_VEL
LIN {X 0,Y 27.645,Z 795.264,A -85,B 0,C 180,E1 -31505.633,E2 -31505.633} C_VEL
LIN {X 0,Y 35.323,Z 785.731,A -85,B 0,C 180,E1 -31505.854,E2 -31505.854} C_VEL
LIN {X 0,Y 42.407,Z 774.905,A -85,B 0,C 180,E1 -31506.101,E2 -31506.101} C_VEL
LIN {X 0,Y 48.603,Z 763.011,A -85,B 0,C 180,E1 -31506.223,E2 -31506.223} C_VEL
LIN {X 0,Y 53.558,Z 750.294,A -85,B 0,C 180,E1 -31506.363,E2 -31506.363} C_VEL
LIN {X 0,Y 57.309,Z 736.579,A -85,B 0,C 180,E1 -31506.489,E2 -31506.489} C_VEL
LIN {X 0,Y 60.131,Z 720.157,A -85,B 0,C 180,E1 -31506.708,E2 -31506.708} C_VEL
LIN {X 0,Y 59.843,Z 716.682,A -85,B 0,C 180,E1 -31510.07,E2 -31510.07} C_VEL
LIN {X 0,Y 59.516,Z 712.055,A -85,B 0,C 180,E1 -31516.512,E2 -31516.512} C_VEL
LIN {X 0,Y 59.474,Z 710.993,A -85,B 0,C 180,E1 -31519.034,E2 -31519.034} C_VEL
LIN {X 0,Y 59.363,Z 711.229,A -85,B 0,C 180,E1 -31524.306,E2 -31524.306} C_VEL
LIN {X 0,Y 59.497,Z 713.654,A -85,B 0,C 180,E1 -31531.401,E2 -31531.401} C_VEL
LIN {X 0,Y 60.013,Z 717.932,A -85,B 0,C 180,E1 -31537.58,E2 -31537.58} C_VEL
LIN {X 0,Y 60.116,Z 718.604,A -85,B 0,C 180,E1 -31538.392,E2 -31538.392} C_VEL
LIN {X 0,Y 57.001,Z 736.348,A -85,B 0,C 180,E1 -31538.66,E2 -31538.66} C_VEL
LIN {X 0,Y 53.574,Z 748.836,A -85,B 0,C 180,E1 -31538.842,E2 -31538.842} C_VEL
LIN {X 0,Y 48.603,Z 761.729,A -85,B 0,C 180,E1 -31538.995,E2 -31538.995} C_VEL
LIN {X 0,Y 42.394,Z 773.836,A -85,B 0,C 180,E1 -31539.215,E2 -31539.215} C_VEL
LIN {X 0,Y 34.768,Z 785.599,A -85,B 0,C 180,E1 -31539.487,E2 -31539.487} C_VEL
LIN {X 0,Y 26.394,Z 795.94,A -85,B 0,C 180,E1 -31539.674,E2 -31539.674} C_VEL
LIN {X 0,Y 17.185,Z 805.25,A -85,B 0,C 180,E1 -31539.932,E2 -31539.932} C_VEL
LIN {X 0,Y 7.124,Z 813.533,A -85,B 0,C 180,E1 -31537.053,E2 -31537.053} C_VEL
LIN {X 0,Y 1.377,Z 817.741,A -85,B 0,C 180,E1 -31499.851,E2 -31499.851} C_VEL
LIN {X 0,Y 3.345,Z 816.542,A -85,B 0,C 180,E1 -31496.564,E2 -31496.564} C_VEL
LIN {X 0,Y 14.087,Z 808.493,A -85,B 0,C 180,E1 -31503.818,E2 -31503.818} C_VEL
LIN {X 0,Y 22.94,Z 800.305,A -85,B 0,C 180,E1 -31505.338,E2 -31505.338} C_VEL
LIN {X 0,Y 27.645,Z 795.264,A -85,B 0,C 180,E1 -31505.633,E2 -31505.633} C_VEL
LIN {X 0,Y 31.264,Z 790.746,A -85,B 0,C 180,E1 -31506.949,E2 -31506.949} C_VEL
LIN {X 0,Y 36.477,Z 782.796,A -85,B 0,C 180,E1 -31511.289,E2 -31511.289} C_VEL
LIN {X 0,Y 41.293,Z 774.315,A -85,B 0,C 180,E1 -31514.691,E2 -31514.691} C_VEL
LIN {X 0,Y 44.108,Z 768.965,A -85,B 0,C 180,E1 -31515.059,E2 -31515.059} C_VEL
LIN {X 0,Y 49.392,Z 757.437,A -85,B 0,C 180,E1 -31514.229,E2 -31514.229} C_VEL
LIN {X 0,Y 53.771,Z 744.497,A -85,B 0,C 180,E1 -31513.702,E2 -31513.702} C_VEL
LIN {X 0,Y 56.763,Z 731.388,A -85,B 0,C 180,E1 -31513.475,E2 -31513.475} C_VEL
LIN {X 0,Y 58.186,Z 722.665,A -85,B 0,C 180,E1 -31513.579,E2 -31513.579} C_VEL
LIN {X 0,Y 58.258,Z 718.466,A -85,B 0,C 180,E1 -31519.244,E2 -31519.244} C_VEL
LIN {X 0,Y 58.287,Z 717.991,A -85,B 0,C 180,E1 -31520.243,E2 -31520.243} C_VEL
LIN {X 0,Y 58.209,Z 718.257,A -85,B 0,C 180,E1 -31523.348,E2 -31523.348} C_VEL
LIN {X 0,Y 58.158,Z 720.165,A -85,B 0,C 180,E1 -31528.902,E2 -31528.902} C_VEL
LIN {X 0,Y 58.191,Z 721.902,A -85,B 0,C 180,E1 -31531.636,E2 -31531.636} C_VEL
LIN {X 0,Y 55.333,Z 737.621,A -85,B 0,C 180,E1 -31531.534,E2 -31531.534} C_VEL
LIN {X 0,Y 51.662,Z 750.616,A -85,B 0,C 180,E1 -31531.21,E2 -31531.21} C_VEL
LIN {X 0,Y 46.423,Z 763.702,A -85,B 0,C 180,E1 -31530.519,E2 -31530.519} C_VEL
LIN {X 0,Y 40.299,Z 775.428,A -85,B 0,C 180,E1 -31529.313,E2 -31529.313} C_VEL
LIN {X 0,Y 33.718,Z 785.62,A -85,B 0,C 180,E1 -31527.645,E2 -31527.645} C_VEL
LIN {X 0,Y 26.101,Z 795.368,A -85,B 0,C 180,E1 -31524.214,E2 -31524.214} C_VEL
LIN {X 0,Y 26.301,Z 795.193,A -85,B 0,C 180,E1 -31520.736,E2 -31520.736} C_VEL
LIN {X 0,Y 34.074,Z 785.328,A -85,B 0,C 180,E1 -31517.464,E2 -31517.464} C_VEL
LIN {X 0,Y 41.063,Z 774.508,A -85,B 0,C 180,E1 -31515.697,E2 -31515.697} C_VEL
LIN {X 0,Y 44.108,Z 768.965,A -85,B 0,C 180,E1 -31515.059,E2 -31515.059} C_VEL
LIN {X 0,Y 46.661,Z 763.641,A -85,B 0,C 180,E1 -31515.457,E2 -31515.457} C_VEL
LIN {X 0,Y 50.126,Z 754.618,A -85,B 0,C 180,E1 -31518.166,E2 -31518.166} C_VEL
LIN {X 0,Y 52.964,Z 745.32,A -85,B 0,C 180,E1 -31520.686,E2 -31520.686} C_VEL
LIN {X 0,Y 54.405,Z 739.557,A -85,B 0,C 180,E1 -31521.009,E2 -31521.009} C_VEL
LIN {X 0,Y 56.848,Z 726.863,A -85,B 0,C 180,E1 -31520.551,E2 -31520.551} C_VEL
LIN {X 0,Y 57.007,Z 725.833,A -85,B 0,C 180,E1 -31520.756,E2 -31520.756} C_VEL
LIN {X 0,Y 57.08,Z 725.256,A -85,B 0,C 180,E1 -31521.673,E2 -31521.673} C_VEL
LIN {X 0,Y 57.005,Z 725.92,A -85,B 0,C 180,E1 -31524.549,E2 -31524.549} C_VEL
LIN {X 0,Y 54.094,Z 740.872,A -85,B 0,C 180,E1 -31524.031,E2 -31524.031} C_VEL
LIN {X 0,Y 51.132,Z 750.989,A -85,B 0,C 180,E1 -31523.232,E2 -31523.232} C_VEL
LIN {X 0,Y 51.249,Z 750.646,A -85,B 0,C 180,E1 -31521.791,E2 -31521.791} C_VEL
LIN {X 0,Y 54.405,Z 739.557,A -85,B 0,C 180,E1 -31521.009,E2 -31521.009} C_VEL
LIN {X 0,Y 54.405,Z 739.557,A -85,B 0,C 180,E1 -31521.009,E2 -31521.009}

QRS_NEXT_CUT()

QRS_NEXT()
QRS_HOME()

END
